(* Logix 5000 project; controller PLC vendor 1 type 14 code 155 rev 30.14; software revision 30.01 *)

TASK MainTask (continuous, watchdog 500 ms) : MainProgram

MODULES
   Local : vendor 1 type 14 code 155 (PointIO 0, rev 30.14)
      Encoder_Conveyor : vendor 1 type 37 code 52 (Ethernet 192.168.100.195, rev 1.1, MotionDiagnostics RPI 1 ms, MotionSync RPI 4 ms)
      Servo_Bridge_Shift : vendor 1 type 37 code 49 (Ethernet 192.168.100.194, rev 7.1, MotionSync RPI 4 ms, MotionDiagnostics RPI 1 ms)
      Rack_0_Slot_2 : 1734-IB8 (PointIO 2, rev 3.1, Input RPI 20 ms)
           Local:2:I.Data.0   // Slot 2 Input 0
           Local:2:I.Data.1   // Slot 2 Input 1
           Local:2:I.Data.2   // Slot 2 Input 2
           Local:2:I.Data.3   // Slot 2 Input 3
           Local:2:I.Data.4   // Slot 2 Input 4
           Local:2:I.Data.5   // Slot 2 Input 5
           Local:2:I.Data.6   // Slot 2 Input 6
           Local:2:I.Data.7   // Slot 2 Input 7
      Rack_0_Slot_3 : 1734-OB8 (PointIO 3, rev 3.1, Output RPI 20 ms)
           Local:3:O.Data.0   // Slot 3 Output 0
           Local:3:O.Data.1   // Slot 3 Output 1
           Local:3:O.Data.2   // Slot 3 Output 2
           Local:3:O.Data.3   // Slot 3 Output 3
           Local:3:O.Data.4   // Slot 3 Output 4
           Local:3:O.Data.5   // Slot 3 Output 5
           Local:3:O.Data.6   // Slot 3 Output 6
           Local:3:O   // Slot 3 Output
      Discrete_IO : Embedded (PointIO 1, rev 30.11, Output RPI 20 ms)
           Local:1:O   // Slot 1 Output
           Local:1:I.Data.0   // Slot 0 Input 0
           Local:1:I.Data.1   // Slot 0 Input 1
           Local:1:I.Data.10   // Slot 0 Input 10
           Local:1:I.Data.11   // Slot 0 Input 11
           Local:1:I.Data.12   // Slot 0 Input 12
           Local:1:I.Data.13   // Slot 0 Input 13
           Local:1:I.Data.14   // Slot 0 Input 14
           Local:1:I.Data.15   // Slot 0 Input 15
           Local:1:I.Data.2   // Slot 0 Input 2
           Local:1:I.Data.3   // Slot 0 Input 3
           Local:1:I.Data.4   // Slot 0 Input 4
           Local:1:I.Data.5   // Slot 0 Input 5
           Local:1:I.Data.6   // Slot 0 Input 6
           Local:1:I.Data.7   // Slot 0 Input 7
           Local:1:I.Data.8   // Slot 0 Input 8
           Local:1:I.Data.9   // Slot 0 Input 9
      Rack_0_Slot_4 : 1734-OB8 (PointIO 4, rev 3.1, Output RPI 20 ms)
           Local:4:O   // Slot 4 Output
END_MODULES

TYPE Axis_MC_R3b :
STRUCT
   Auto_Enable : BOOL;
   Direction_Fwd : BOOL;
   Direction_Rev : BOOL;
   Direction_Fwd_DINT : DINT;
   Direction_Rev_DINT : DINT;
   Multiplier_Distance : REAL;
   Multiplier_Speed : REAL;
   Multiplier_Acc_Dec : REAL;
   Distance_Home_Offset : REAL;
   Distance_Row_to_Row : REAL;
   Distance_First_Row : REAL;
   Distance_Flight_to_Flight : REAL;
   Number_of_Rows : REAL;
   Speed_Homing : REAL;
   Speed_Jog_FWD : REAL;
   Speed_Jog_REV : REAL;
   Speed_Prime : REAL;
   Speed_Cleaning : REAL;
   Speed_Auto_FWD : REAL;
   Speed_Auto_REV : REAL;
   Accel_Homing : REAL;
   Accel_Jog : REAL;
   Accel_Prime : REAL;
   Accel_Auto : REAL;
   Accel_Raw : REAL;
   Accel_Scaled : REAL;
   Decel_Estop : REAL;
   Decel_Homing : REAL;
   Decel_Jog : REAL;
   Decel_Prime : REAL;
   Decel_Auto : REAL;
   Decel_Raw : REAL;
   Decel_Scaled : REAL;
   Status_Faulted : BOOL;
   Status_Fault_Code : DINT;
   Status_Homed : BOOL;
   Status_Homing : BOOL;
   Status_Raw_Position : DINT;
   Status_Scaled_Position : REAL;
   Status_Jogging : BOOL;
   Status_Jogging_Stopped_OS : BOOL;
   Status_In_Motion : BOOL;
   Status_In_Motion_OS : BOOL;
   Status_Stopped : BOOL;
   Status_Stopped_OS : BOOL;
   Status_Safe_to_Move : BOOL;
   HMI_PB_Jog_FWD : BOOL;
   HMI_PB_Jog_REV : BOOL;
   Jog_FWD : BOOL;
   Jog_REV : BOOL;
   Jog_FWD_OS : BOOL;
   Jog_REV_OS : BOOL;
   HMI_PB_Home_Servo : BOOL;
   HMI_PB_Home_Servo_OS : BOOL;
   Homing_Needed_Next_Move : BOOL;   // Registration needed during next long move
   Homing_Needed_Now : BOOL;   // Registration needed after e-stop
   Homing_Counter : COUNTER;   // Registration counter for cycles before homing or registration needed
   Homing_Counter_DN_OS : BOOL;
   Homing_Timer_Step : TIMER[10];
   Homing_Sensor_Active_OS : BOOL;
   Homing_Sensor_Deactive_OS : BOOL;
   Homing_Failure : BOOL;
   Timer_Jog_FWD_Delay : TIMER;
   Timer_Jog_REV_Delay : TIMER;
   Timer_Servo_Safe_to_Move : TIMER;
   Overtravel_Fwd_Active_OS : BOOL;
   Overtravel_Fwd_Deactive_OS : BOOL;
   Overtravel_Rev_Active_OS : BOOL;
   Overtravel_Rev_Deactive_OS : BOOL;
   Overtravel_Front_Active_OS : BOOL;
   Overtravel_Front_Deactive_OS : BOOL;
   Overtravel_Rear_Active_OS : BOOL;
   Overtravel_Rear_Deactive_OS : BOOL;
   Cam_M_Offset : DINT;
   Cam_S_Offset : DINT;
   Cam_M_Scaling : DINT;
   Cam_S_Scaling : DINT;
   OS : DINT[2];
   MSO : MOTION_INSTRUCTION;
   MSF : MOTION_INSTRUCTION;
   MASR : MOTION_INSTRUCTION;
   MAFR : MOTION_INSTRUCTION;
   MAJ : MOTION_INSTRUCTION[10];
   MAJ_DIRECTION : DINT[10];
   MAJ_SPEED : REAL[10];
   MAJ_ACC : REAL[10];
   MAJ_DEC : REAL[10];
   MAM : MOTION_INSTRUCTION[10];
   MAM_TYPE : DINT[10];
   MAM_DISTANCE : REAL[10];
   MAM_SPEED : REAL[10];
   MAM_ACC : REAL[10];
   MAM_DEC : REAL[10];
   MAS : MOTION_INSTRUCTION[10];
   MAS_DEC : REAL[10];
   MAH : MOTION_INSTRUCTION[5];
   MCD : MOTION_INSTRUCTION[10];
   MRP : MOTION_INSTRUCTION;
   MGS : MOTION_INSTRUCTION;
   MGSD : MOTION_INSTRUCTION;
   MGSR : MOTION_INSTRUCTION;
   MGSP : MOTION_INSTRUCTION;
   MAG : MOTION_INSTRUCTION[5];
   MAG_DIRECTION : DINT[5];
   MAG_TYPE : DINT[5];
   MAG_DISTANCE : REAL[5];
   MAG_SPEED : REAL[5];
   MAG_ACC : REAL[5];
   MAG_DEC : REAL[5];
   MAG_RATIO : REAL[5];
   MAG_S_COUNTS : DINT[5];
   MAG_M_COUNTS : DINT[5];
END_STRUCT
END_TYPE

TYPE Denester_R2b :
STRUCT
   HMI_Auger_VFD_Jog : BOOL;
   HMI_Trigger : BOOL;
   HMI_Trigger_OS : BOOL;
   Trigger : BOOL;
   Trigger_OS : BOOL;
   Auger_Direction_Fwd : BOOL;
   Auger_Direction_Rev : BOOL;
   Auger_VFD_Run : BOOL;
   Auger_VFD_Jog : BOOL;
   Auger_VFD_Speed_Auto : REAL;
   Auger_VFD_Speed_Jog : REAL;
   Auger_Prox_OS : BOOL;
   Status_Ready : BOOL;
   Status_Done : BOOL;
   Status_Done_OS : BOOL;
   Timer_Auger_Run_Delay : TIMER;
   Low_Cups_OS : BOOL;
   Low_Cups_Warning : BOOL;
   Timer_Trigger_Delay : TIMER;
   Timer_Trigger_Duration : TIMER;
   OS : DINT;
END_STRUCT
END_TYPE

TYPE Depositor_R2b :
STRUCT
   HMI_Trigger_Deposit : BOOL;
   HMI_Trigger_Deposit_OS : BOOL;
   Prime_Trigger_Deposit_OS : BOOL;
   Trigger_Deposit : BOOL;
   Trigger_Deposit_OS : BOOL;
   Piston_Deposit : DINT;   // Product Piston deposit
   Piston_Suction : DINT;   // Product Piston suction
   Product_Valve_Deposit : DINT;   // Product Valve deposit position
   Spout_Open : DINT;   // Open Spout
   Dive_Down : DINT;
   Dive_Up : DINT;
   Status_Suction_Complete : BOOL;
   Status_Suction_Complete_OS : BOOL;
   Status_Deposit_Complete : BOOL;
   Status_Deposit_Complete_OS : BOOL;
   Status_Done : BOOL;
   Status_Done_OS : BOOL;
   Status_Ready : BOOL;
   Timer_Blowoff_Delay : TIMER;
   Timer_Blowoff_Duration : TIMER;
   Timer_Dive_Delay : TIMER;
   Timer_Dive_Duration : TIMER;
   Timer_Dive_Timeout : TIMER;
   Timer_Trigger_Duration : TIMER;
   Timer_Trigger_Delay : TIMER;
   Timer_Prime : TIMER;
   Timer_Shift_Delay_Suction : TIMER;
   Timer_Shift_Delay_Deposit : TIMER;
   Timer_Spout_Timeout : TIMER;
   OS : DINT;
END_STRUCT
END_TYPE

TYPE Forces_R2b :
STRUCT
   DI_0 : DINT;   // INPUT FORCE
   DI_1 : DINT;   // INPUT FORCE
   DI_2 : DINT;   // INPUT FORCE
   DI_3 : DINT;   // INPUT FORCE
   DI_4 : DINT;   // INPUT FORCE
   DI_5 : DINT;   // INPUT FORCE
   DO_0 : DINT;   // OUTPUT FORCE
   DO_1 : DINT;   // OUTPUT FORCE
   DO_2 : DINT;   // OUTPUT FORCE
   DO_3 : DINT;   // OUTPUT FORCE
   DO_4 : DINT;   // OUTPUT FORCE
   DO_5 : DINT;   // OUTPUT FORCE
   DO_6 : DINT;   // OUTPUT FORCE
   DO_7 : DINT;   // OUTPUT FORCE
   DO_8 : DINT;   // OUTPUT FORCE
   DO_9 : DINT;   // OUTPUT FORCE
   DO_10 : DINT;   // OUTPUT FORCE
   R_DO_0 : DINT;   // OUTPUT FORCE
   R_DO_1 : DINT;   // OUTPUT FORCE
   R_DO_2 : DINT;   // OUTPUT FORCE
   R_DO_3 : DINT;   // OUTPUT FORCE
   R_DO_4 : DINT;   // OUTPUT FORCE
   R_DO_5 : DINT;   // OUTPUT FORCE
END_STRUCT
END_TYPE

TYPE IO_R2a :
STRUCT
   DI_0 : DINT;
   DI_1 : DINT;
   DI_2 : DINT;
   DI_3 : DINT;
   DI_4 : DINT;
   DI_5 : DINT;
   DI_6 : DINT;
   DI_7 : DINT;
   DI_8 : DINT;
   DI_9 : DINT;
   DI_10 : DINT;
   DO_0 : DINT;
   DO_1 : DINT;
   DO_2 : DINT;
   DO_3 : DINT;
   DO_4 : DINT;
   DO_5 : DINT;
   DO_6 : DINT;
   DO_7 : DINT;
   DO_8 : DINT;
   DO_9 : DINT;
   DO_10 : DINT;
   R_DI_0 : DINT;
   R_DI_1 : DINT;
   R_DI_2 : DINT;
   R_DI_3 : DINT;
   R_DI_4 : DINT;
   R_DI_5 : DINT;
   R_DO_0 : DINT;
   R_DO_1 : DINT;
   R_DO_2 : DINT;
   R_DO_3 : DINT;
   R_DO_4 : DINT;
   R_DO_5 : DINT;
END_STRUCT
END_TYPE

TYPE Login_R2a :
STRUCT
   User : DINT;
   User_Logged_In : DINT;
   User_New : DINT;
   User_Active : BOOL;
   No_Access : BOOL;
   Password_Entered : DINT;
   Password_New : DINT;
   Password_Old : DINT;
   Password_Admin : DINT;
   Password_Maint : DINT;
   Password_Lead : DINT;
   Password_HBTech : DINT;
   Password_Temp : DINT;
   Password_Backdoor : DINT;
   Password_Oper : DINT;
   PB_Reset_Passwords : BOOL;
   PB_Change_Password : BOOL;
   PB_Change_Password_Yes : BOOL;
   PB_Change_Password_No : BOOL;
   PB_Logout : BOOL;
   Auto_Logout_Minutes : INT;
   Timer_Auto_Logout : TIMER;
   Timer_Reset_Delay : TIMER;
   Timer_Password_Change_Confirm : TIMER;
   Timer_Password_Change_Timeout : TIMER;
   Visible_New_Password : BOOL;
   Visible_Change_Password : BOOL;
   Visible_Change_Confirm : BOOL;
   Visible_Password_Changed : BOOL;
END_STRUCT
END_TYPE

TYPE NCNF_Arrays_R2a :
STRUCT
   Bitshift : DINT[4];
END_STRUCT
END_TYPE

TYPE NCNF_R2a :
STRUCT
   Flight_Detect_OS_Rising : BOOL;   // FLIGHT DETECT RISING OS
   Flight_Detect_OS_Falling : BOOL;   // FLIGHT DETECT FALLING OS
   Target_Detected : BOOL[32];   // NC/NF TARGET DETECTED
   Lane : NCNF_Arrays_R2a[10];   // NC/NF BITSHIFTS
   Bitshift_Control : CONTROL[10];   // NC/NF BITSHIFT CONTROLS
   HMI_PB_Reset : BOOL;   // NC/NF HMI BITSHIFT RESET
   HMI_PB_Fill : BOOL;   // NC/NF HMI BITSHIFT FILL
   HMI_PB_Bypass : BOOL;   // NC/NF HMI BITSHIFT BYPASS
   Timer_Flight_Detect_OFF : TIMER;
END_STRUCT
END_TYPE

TYPE Rates_R2b :
STRUCT
   HMI_PB_Reset_Counter : BOOL;
   Counter_Cycle : COUNTER;
   Counter_Total : COUNTER;
   Timer_CPM_Minute : TIMER;
   Timer_CPM_Seconds : DINT;
   Timer_Cycle_Time : TIMER;
   Cycle_Time : DINT;
   CPM_Current : DINT;
   CPM_Previous : DINT;
   PPM_Current : DINT;
   PPM_Previous : DINT;
   Rows_Per_Pan : DINT;
   Total_Count : DINT;
END_STRUCT
END_TYPE

TYPE Recipe_R2c :
STRUCT
   Active_Recipe_Num : DINT;
   Active_Recipe_Name : STRING;
   Active_Recipe : DINT[15];
   Selected_Recipe_Num : DINT;
   Selected_Recipe_Name : STRING;
   Selected_Recipe : DINT[15];
   Selected_Recipe_Edit_Num : DINT;
   Previous_Selected_Recipe_Num : DINT;
   Indirect_Recipe_Selected : DINT;
   Indirect_Recipe_Selected_Edit : DINT;
   Recipe_Changed_OS : BOOL;
   Load_Selected_Recipe_Num : DINT;
   Saveas_Source_Recipe_Num : DINT;
   Saveas_Target_Recipe_Num : DINT;
   HMI_PB_Load : BOOL;
   HMI_PB_Save : BOOL;
   HMI_PB_Saveas : BOOL;
   HMI_PB_Rename : BOOL;
   Timer_Load : TIMER;
   Timer_Save : TIMER;
   Timer_Saveas : TIMER;
   Names_Pointer : DINT;
   Names_Pointer_Temp : DINT;
   Names_New_Name : STRING;
   Names_Old_Name : STRING;
END_STRUCT
END_TYPE

TYPE Sequencer_R2a :
STRUCT
   Step : DINT;   // Current Step
   Step_OS : BOOL[256];   // Current Step OS
   Timer : TIMER[256];   // Current Step Timer
   OS : BOOL[256];   // OS
END_STRUCT
END_TYPE

TYPE System_R2e :   // System
STRUCT
   HMI_Current_Screen : DINT;
   HMI_Forced_Screen : DINT;
   HMI_PB_Estop_Reset : BOOL;
   HMI_PB_Start : BOOL;
   HMI_PB_Stop : BOOL;
   HMI_PB_Prime : BOOL;
   HMI_PB_Prime_OS : BOOL;
   HMI_PB_Auto : BOOL;
   HMI_PB_Auto_OS : BOOL;
   HMI_PB_Clean : BOOL;
   HMI_PB_Clean_OS : BOOL;
   HMI_PB_Clear_Alarms : BOOL;
   HMI_PB_Silence_Alarms : BOOL;
   HMI_PB_Home_Servos : BOOL;
   HMI_PB_Home_Servos_OS : BOOL;
   HMI_PB_Off : BOOL;
   HMI_PB_Off_OS : BOOL;
   HMI_PB_Wipe_Screen_Reset : BOOL;
   HMI_PB_Recipe_Initialize : BOOL;
   HMI_Visible_PB : BOOL;
   HMI_Visible_Estop_Reset : BOOL;
   HMI_Visible_Home_Servos : BOOL;
   HMI_Visible_Clear_Alarms : BOOL;
   HMI_Visible_Silence_Alarms : BOOL;
   Local_PB_Start : BOOL;
   Local_PB_Stop : BOOL;
   Local_Estop_Reset : BOOL;
   Estop_Reset_Enabled : BOOL;
   Timer_Starting : TIMER;
   Timer_Starting_TT_OS : BOOL;
   Timer_Starting_DN_OS : BOOL;
   Timer_Stopping : TIMER;
   Timer_Stopping_EN_OS : BOOL;
   Timer_Stopping_DN_OS : BOOL;
   Timer_Estop_Not_OK : TIMER;
   Timer_Estop_Not_OK_TT_OS : BOOL;
   Timer_Estop_Not_OK_DN_OS : BOOL;
   Timer_EStop_Reset : TIMER;
   Timer_Estop_OK : TIMER;
   Timer_Estop_OK_TT_OS : BOOL;
   Timer_Estop_OK_DN_OS : BOOL;
   Timer_Power_Up : TIMER;
   Timer_Power_Up_OS : BOOL;
   Timer_Alarm_Timeout : TIMER;
   Timer_Alarm_Timeout_OS : BOOL;
   Timer_Flasher_Slow_On : TIMER;
   Timer_Flasher_Slow_Off : TIMER;
   Timer_Flasher_Fast_On : TIMER;
   Timer_Flasher_Fast_Off : TIMER;
   Timer_Servos_Home : TIMER;
   Timer_Alarm_Horn : TIMER;
   Timer_Wipe_Screen : TIMER;
   Timer_Screen_Force : TIMER;
   Mode_Auto : BOOL;
   Mode_Off : BOOL;
   Mode_Prime : BOOL;
   Mode_Clean : BOOL;
   Mode_Integer : DINT;
   Mode_Changed_OS : BOOL;
   Status_EStop_Active : BOOL;
   Status_Estop_OK : BOOL;
   Status_Estop_OK_OS : BOOL;
   Status_Estop_NOT_OK : BOOL;
   Status_Estop_NOT_OK_OS : BOOL;
   Status_Alarm : BOOL;
   Status_Alarm_OS : BOOL;
   Status_New_Alarm : BOOL;
   Status_Warning : BOOL;
   Status_DINT : DINT;   // \
   Servos_Home : BOOL;
   Servos_Home_OS : BOOL;
   Servos_Homed : BOOL;
   Servos_Homed_OS : BOOL;
   Servos_Homing_Requested : BOOL;
   Servos_Homing : BOOL;
   Servos_Homing_OS : BOOL;
   Servos_OK : BOOL;
   Always_ON_Bit : BOOL;
   Always_OFF_Bit : BOOL;
   Test_Bits : DINT;
   Comms_Scan_Timer : TIMER;
   Comms_Scan_Counter : DINT;
END_STRUCT
END_TYPE

VAR_GLOBAL   (* controller tags *)
   Alarm_Timer : TIMER[2,32] := ([0,1].PRE := 1000, [0,2].PRE := 5, [0,3].PRE := 5, [0,4].PRE := 5, [0,5].PRE := 10, [0,6].PRE := 100, [0,7].PRE := 500, [0,8].PRE := 5000, [0,9].PRE := 7500, [0,10].PRE := 500, [0,11].PRE := 20000, [0,12].PRE := 5, [0,13].PRE := 5, [0,14].PRE := 5, [0,15].PRE := 5, [0,16].PRE := 5, [0,17].PRE := 1000, [0,18].PRE := 2000, [0,19].PRE := 100, [0,20].PRE := 20000, [0,21].PRE := 20000, [0,22].PRE := 100, [0,23].PRE := 100);
   Alarm_Word_Compare : DINT[3];
   Alarm_Word_Current : DINT[3];
   Alarm_Word_New : DINT[3];
   Alarm_Word_Previous : DINT[3];
   always_open : BOOL;
   Bridge_Timer_Gearing_Delay : TIMER := (PRE := 30);
   Bridge_Timer_Gearing_Delay_DN_OS : BOOL;
   Bridge_Timer_Gearing_Duration : TIMER;
   Bridge_Timer_Gearing_Duration_DN_OS : BOOL;
   Bypass_Encoder : BOOL;
   Denester : Denester_R2b := (Timer_Trigger_Delay.PRE := 5, Timer_Trigger_Duration.PRE := 40);
   Denester_Flight_Counter : COUNTER := (PRE := 1);
   Denester_index_counter : COUNTER := (PRE := 4, ACC := 2);
   Depositor : Depositor_R2b := (Timer_Blowoff_Delay.PRE := 20, Timer_Blowoff_Duration.PRE := 200, Timer_Dive_Delay.PRE := 5, Timer_Dive_Duration.PRE := 1095, Timer_Trigger_Delay.PRE := 25, Timer_Prime.PRE := 1000, Timer_Spout_Timeout.PRE := 1500);
   Depositor_Bridge_Up : BOOL;
   Encoder_Conveyor : AXIS_CIP_DRIVE;
   equal_to_20 : BOOL;
   FORCE_GO_SIGNAL : BOOL;
   FORCE_TRIGGER : BOOL;
   Forces : Forces_R2b := (DO_3 := 8);
   HMI_Enable_Denester : BOOL := 1;
   homing_timeout : TIMER := (PRE := 20000);
   IO : IO_R2a := (DI_1 := 33228, DI_2 := 32, DO_1 := 34, DO_3 := 8);
        .DI_2.0   // SPARE
        .DI_2.1   // BRIDGE UP PROX
        .DI_2.2   // BRIDGE OVERTRAVEL PROX
        .DI_2.3   // BRIDGE HOME PROX
        .DI_2.4   // SPARE
        .DI_2.5   // SPARE
        .DI_2.6   // SPARE
        .DI_2.7   // SPARE
        .DO_1.0   // STACK LIGHT HORN
        .DO_1.1   // STACK LIGHT GREEN
        .DO_1.10   // FILLER SPOUT #3 TRIGGER
        .DO_1.11   // FILLER SPOUT #4 TRIGGER
        .DO_1.12   // FILLER SPOUT #5 TRIGGER
        .DO_1.13   // FILLER SPOUT #6 TRIGGER
        .DO_1.14   // FILLER SPOUT #7 TRIGGER
        .DO_1.15   // FILLER SPOUT #8 TRIGGER
        .DO_1.2   // STACK LIGHT AMBER
        .DO_1.3   // STACK LIGHT RED
        .DO_1.4   // DONE SIGNAL TO CUSTOMER
        .DO_1.5   // PLC E-STOP RESET
        .DO_1.6   // READY SIGNAL TO CUSTOMER
        .DO_1.7   // DENESTER TRIGGER
        .DO_1.8   // FILLER SPOUT #1 TRIGGER
        .DO_1.9   // FILLER SPOUT #2 TRIGGER
        .DO_3.0   // BRIDGE DOWN SPOUTS #1-4
        .DO_3.1   // BRIDGE UP SPOUTS #1-4
        .DO_3.2   // BLOWOFF SPOUTS #1-4
        .DO_3.3   // SPOUT #1 OPEN
        .DO_3.4   // SPOUT #2 OPEN
        .DO_3.5   // SPOUT #3 OPEN
        .DO_3.6   // SPOUT #4 OPEN
        .DO_3.7   // SPARE
        .DO_4.0   // BRIDGE DOWN SPOUTS #5-8
        .DO_4.1   // BRIDGE UP SPOUTS #5-8
        .DO_4.2   // BLOWOFF SPOUTS #5-8
        .DO_4.3   // SPOUT #5 OPEN
        .DO_4.4   // SPOUT #6 OPEN
        .DO_4.5   // SPOUT #7 OPEN
        .DO_4.6   // SPOUT #8 OPEN
        .DO_4.7   // SPARE
        .DI_1.0   // SPARE
        .DI_1.1   // SPARE
        .DI_1.10   // FILLER PRIME MODE ACTIVE
        .DI_1.11   // E-STOP PRESSED 1-HOLE UPSTREAM
        .DI_1.12   // ULMA GO SIGNAL/ FLIGHT DETECT
        .DI_1.13   // ULMA RUNNING RELAY
        .DI_1.14   // NC/NF SENSOR LANE #0
        .DI_1.15   // NC/NF SENSOR LANE #1
        .DI_1.2   // AIR PRESSURE SWITCH
        .DI_1.3   // E-STOP OK
        .DI_1.4   // E-STOP PRESSED MAIN
        .DI_1.5   // E-STOP PRESSED 1-HOLE DOWNSTREAM
        .DI_1.6   // UPSTREAM DOOR
        .DI_1.7   // DOWNSTREAM DOOR
        .DI_1.8   // DOCKING SAFETY SENSOR
        .DI_1.9   // FILLER DONE/READY
   Login : Login_R2a := (Password_Admin := 111, Password_Maint := 222, Password_Lead := 333, Password_HBTech := 32767, Password_Temp := 555, Password_Backdoor := 80808, Password_Oper := 444, Auto_Logout_Minutes := 60, Timer_Auto_Logout.PRE := 3600000);
        .User   // Login User 1 = ADMIN 2 = MAINT 3 = LEAD 4 = OPER 5 = TEMP 6 = BACKDOOR 7 = HBTECH
        .User_Logged_In   // Login User Logged In
        .Password_Entered   // Login Password Entered
   MV_conveyor_moving : BOOL;
   MV_conveyor_stopped : BOOL;
   MV_Encoder_Stop_Threshold : DINT;
   MV_Encoder_Stop_Value : REAL := 0.3;
   MV_Encoder_Stop_Value2 : REAL := 0.2;
   mv_index_counter : COUNTER := (PRE := 15, ACC := 5);
   MV_indexes : DINT := 4;
   MV_Rate : DINT := 100;
   MV_total_indexes : COUNTER := (PRE := 100, ACC := 343, DN := 1);
   NC_NF : NCNF_R2a := (Target_Detected[1] := 1, Lane[0].Bitshift[0] := 2147483647, Lane[0].Bitshift[1] := 2147483647, Lane[0].Bitshift[2] := 2147483647, Lane[0].Bitshift[3] := 2147483647, Lane[1].Bitshift[0] := 2147483647, Lane[1].Bitshift[1] := 2147483647, Lane[1].Bitshift[2] := 2147483647, Lane[1].Bitshift[3] := 2147483647, Bitshift_Control[0].LEN := 4, Bitshift_Control[0].UL := 1, Bitshift_Control[1].LEN := 4, Bitshift_Control[1].UL := 1, HMI_PB_Bypass := 1);   // NC/NF BITSHIFTS
        .Flight_Detect_OS_Rising   // Flight Detect One Shot Rising
        .Flight_Detect_OS_Falling   // Flight Detect One Shot Falling
   OS : INT[10] := ([0] := 268, [1] := 42, [2] := 28356, [3] := 2114, [4] := 6176, [5] := 19966, [6] := -32768);
        [0].15   // DUMMY TEST BIT
        [2].2   // SUTEY
        [2].5   // TEST BIT
        [3].13   // IGNORE
        [2].3   // SUTEY
        [5].0   // OS to position Bridge for CIP
        [7].0   // TEST BIT
        [3].2   // SUTEY
   Rates : Rates_R2b := (Counter_Cycle.PRE := 1000, Counter_Total.PRE := 10000000, Counter_Total.ACC := 701468, Timer_CPM_Minute.PRE := 60000, Timer_CPM_Minute.ACC := 3755, Timer_CPM_Minute.EN := 1, Timer_CPM_Minute.TT := 1, Timer_CPM_Seconds := 3, Timer_Cycle_Time.ACC := 1, Timer_Cycle_Time.EN := 1, Timer_Cycle_Time.DN := 1, Cycle_Time := 1);
   Recipe : Recipe_R2c := (Selected_Recipe_Num := 1, Selected_Recipe_Edit_Num := 22, Previous_Selected_Recipe_Num := 1);
        .Active_Recipe[0].0   // Active Recipe VFD Conveyor ON/OFF
   Recipe_Names : STRING[23] := ([1] := ' 2ZOG AU', [2] := 'ERICEP2 ', [3] := 'ERICEP3 ', [4] := 'ERICEP4 ', [5] := 'ERICEP5 ', [6] := 'ERICEP6 ', [7] := 'ERICEP7 ', [8] := 'ERICEP8 ', [9] := 'ERICEP9 ', [10] := 'ERICEP1  0', [11] := 'ERICEP1  1', [12] := 'ERICEP1  2', [13] := 'ERICEP1  3', [14] := 'ERICEP1  4', [15] := 'ERICEP1  5', [16] := 'ERICEP1  6', [17] := 'ERICEP1  7', [18] := 'ERICEP1  8', [19] := 'ERICEP1  9', [20] := 'ERICEP2  0', [21] := 'ETTS', [22] := 'ETTS');
   Recipe_Setpoints_DINT : DINT[23,20] := ([0,0] := 55, [0,1] := 56, [0,2] := 56, [0,3] := 15, [0,7] := 51, [0,8] := 60, [0,12] := 52, [0,13] := 60, [1,0] := 63, [1,1] := 56, [1,2] := 56, [1,3] := 15, [1,7] := 51, [1,8] := 60, [1,12] := 52, [1,13] := 60, [2,0] := 63, [2,1] := 56, [2,2] := 56, [2,3] := 15, [2,7] := 51, [2,8] := 60, [2,12] := 52, [2,13] := 60, [3,0] := 63, [3,1] := 56, [3,2] := 56, [3,3] := 15, [3,7] := 51, [3,8] := 60, [3,12] := 52, [3,13] := 60, [4,0] := 63, [4,1] := 56, [4,2] := 56, [4,3] := 15, [4,7] := 51, [4,8] := 60, [4,12] := 52, [4,13] := 60, [5,0] := 63, [5,1] := 56, [5,2] := 56, [5,3] := 15, [5,7] := 51, [5,8] := 60, [5,12] := 52, [5,13] := 60, [6,0] := 63, [6,1] := 56, [6,2] := 56, [6,3] := 15, [6,7] := 51, [6,8] := 60, [6,12] := 52, [6,13] := 60, [7,0] := 63, [7,1] := 56, [7,2] := 56, [7,3] := 15,
        [7,7] := 51, [7,8] := 60, [7,12] := 52, [7,13] := 60, [8,0] := 63, [8,1] := 56, [8,2] := 56, [8,3] := 15, [8,7] := 51, [8,8] := 60, [8,12] := 52, [8,13] := 60, [9,0] := 63, [9,1] := 56, [9,2] := 56, [9,3] := 15, [9,7] := 51, [9,8] := 60, [9,12] := 52, [9,13] := 60, [10,0] := 63, [10,1] := 56, [10,2] := 56, [10,3] := 15, [10,7] := 51, [10,8] := 60, [10,12] := 52, [10,13] := 60, [11,0] := 63, [11,1] := 56, [11,2] := 56, [11,3] := 15, [11,7] := 51, [11,8] := 60, [11,12] := 52, [11,13] := 60, [12,0] := 63, [12,1] := 56, [12,2] := 56, [12,3] := 15, [12,7] := 51, [12,8] := 60, [12,12] := 52, [12,13] := 60, [13,0] := 63, [13,1] := 56, [13,2] := 56, [13,3] := 15, [13,7] := 51, [13,8] := 60, [13,12] := 52, [13,13] := 60, [14,0] := 63, [14,1] := 56, [14,2] := 56, [14,3] := 15, [14,7] := 51, [14,8] := 60, [14,12] := 52, [14,13] := 60,
        [15,0] := 63, [15,1] := 56, [15,2] := 56, [15,3] := 15, [15,7] := 51, [15,8] := 60, [15,12] := 52, [15,13] := 60, [16,0] := 63, [16,1] := 56, [16,2] := 56, [16,3] := 15, [16,7] := 51, [16,8] := 60, [16,12] := 52, [16,13] := 60, [17,0] := 63, [17,1] := 56, [17,2] := 56, [17,3] := 15, [17,7] := 51, [17,8] := 60, [17,12] := 52, [17,13] := 60, [18,0] := 63, [18,1] := 56, [18,2] := 56, [18,3] := 15, [18,7] := 51, [18,8] := 60, [18,12] := 52, [18,13] := 60, [19,0] := 63, [19,1] := 56, [19,2] := 56, [19,3] := 15, [19,7] := 51, [19,8] := 60, [19,12] := 52, [19,13] := 60, [20,0] := 63, [20,1] := 56, [20,2] := 56, [20,3] := 15, [20,7] := 51, [20,8] := 60, [20,12] := 52, [20,13] := 60, [21,0] := 63, [21,1] := 56, [21,2] := 56, [21,3] := 15, [21,7] := 51, [21,8] := 60, [21,12] := 52, [21,13] := 60, [22,0] := 63, [22,1] := 56, [22,2] := 56, [22,3] := 15,
        [22,7] := 51, [22,8] := 60, [22,12] := 52, [22,13] := 60);
        [0,0]   // Recipe Bools
        [0,0].0   // Recipe Depositor On/Off
        [0,0].1   // Recipe Bridge Dive On/Off
        [0,0].2   // Recipe Bridge Shift On/Off
        [0,0].3   // Recipe Blowoff On/Off
        [0,0].4   // Recipe Orbit B On/Off
        [0,0].5   // Recipe Filler A On/Off
        [0,0].6   // Filler A Level Control On/Off
        [0,0].7   // Filler B Level Control On/Off
        [0,12]   // Filler B Suction Velocity
        [0,13]   // Filler B Deposit Velocity
        [0,1]   // Flighted Conveyor Speed
        [0,2]   // Overrrunning Conveyor Speed
        [0,7]   // Filler A Suction Velocity
        [0,8]   // Filler A Deposit Velocity
   Recipe_Setpoints_DINT_Temp : DINT[20] := ([0] := 63, [1] := 56, [2] := 56, [3] := 15, [7] := 51, [8] := 60, [12] := 52, [13] := 60);
   Recipe_Setpoints_REAL : REAL[23,20] := ([0,0] := 5.0, [0,1] := 0.7, [0,2] := 20.0, [0,3] := 200.0, [0,4] := 5.0, [0,5] := 1095.0, [0,6] := 51.0, [0,8] := 100.0, [0,9] := 200.0, [0,10] := 5.0, [0,14] := 7.5, [0,15] := 10.0, [1,0] := 5.0, [1,1] := 0.7, [1,2] := 400.0, [1,3] := 75.0, [1,4] := 5.0, [1,5] := 800.0, [1,6] := 51.0, [1,8] := 100.0, [1,9] := 200.0, [1,14] := 7.5, [1,15] := 10.0, [2,0] := 5.0, [2,1] := 0.7, [2,2] := 400.0, [2,3] := 75.0, [2,4] := 5.0, [2,5] := 800.0, [2,6] := 51.0, [2,8] := 100.0, [2,9] := 200.0, [2,14] := 7.5, [2,15] := 10.0, [3,0] := 5.0, [3,1] := 0.7, [3,2] := 400.0, [3,3] := 75.0, [3,4] := 5.0, [3,5] := 800.0, [3,6] := 51.0, [3,8] := 100.0, [3,9] := 200.0, [3,14] := 7.5, [3,15] := 10.0, [4,0] := 5.0, [4,1] := 0.7, [4,2] := 400.0, [4,3] := 75.0, [4,4] := 5.0, [4,5] := 800.0, [4,6] := 51.0, [4,8] := 100.0, [4,9] := 200.0, [4,14] := 7.5, [4,15] := 10.0, [5,0] := 5.0, [5,1] := 0.7, [5,2] := 400.0, [5,3] := 75.0,
        [5,4] := 5.0, [5,5] := 800.0, [5,6] := 51.0, [5,8] := 100.0, [5,9] := 200.0, [5,14] := 7.5, [5,15] := 10.0, [6,0] := 5.0, [6,1] := 0.7, [6,2] := 400.0, [6,3] := 75.0, [6,4] := 5.0, [6,5] := 800.0, [6,6] := 51.0, [6,8] := 100.0, [6,9] := 200.0, [6,14] := 7.5, [6,15] := 10.0, [7,0] := 5.0, [7,1] := 0.7, [7,2] := 400.0, [7,3] := 75.0, [7,4] := 5.0, [7,5] := 800.0, [7,6] := 51.0, [7,8] := 100.0, [7,9] := 200.0, [7,14] := 7.5, [7,15] := 10.0, [8,0] := 5.0, [8,1] := 0.7, [8,2] := 400.0, [8,3] := 75.0, [8,4] := 5.0, [8,5] := 800.0, [8,6] := 51.0, [8,8] := 100.0, [8,9] := 200.0, [8,14] := 7.5, [8,15] := 10.0, [9,0] := 5.0, [9,1] := 0.7, [9,2] := 400.0, [9,3] := 75.0, [9,4] := 5.0, [9,5] := 800.0, [9,6] := 51.0, [9,8] := 100.0, [9,9] := 200.0, [9,14] := 7.5, [9,15] := 10.0, [10,0] := 5.0, [10,1] := 0.7, [10,2] := 400.0, [10,3] := 75.0, [10,4] := 5.0, [10,5] := 800.0, [10,6] := 51.0, [10,8] := 100.0, [10,9] := 200.0,
        [10,14] := 7.5, [10,15] := 10.0, [11,0] := 5.0, [11,1] := 0.7, [11,2] := 400.0, [11,3] := 75.0, [11,4] := 5.0, [11,5] := 800.0, [11,6] := 51.0, [11,8] := 100.0, [11,9] := 200.0, [11,14] := 7.5, [11,15] := 10.0, [12,0] := 5.0, [12,1] := 0.7, [12,2] := 400.0, [12,3] := 75.0, [12,4] := 5.0, [12,5] := 800.0, [12,6] := 51.0, [12,8] := 100.0, [12,9] := 200.0, [12,14] := 7.5, [12,15] := 10.0, [13,0] := 5.0, [13,1] := 0.7, [13,2] := 400.0, [13,3] := 75.0, [13,4] := 5.0, [13,5] := 800.0, [13,6] := 51.0, [13,8] := 100.0, [13,9] := 200.0, [13,14] := 7.5, [13,15] := 10.0, [14,0] := 5.0, [14,1] := 0.7, [14,2] := 400.0, [14,3] := 75.0, [14,4] := 5.0, [14,5] := 800.0, [14,6] := 51.0, [14,8] := 100.0, [14,9] := 200.0, [14,14] := 7.5, [14,15] := 10.0, [15,0] := 5.0, [15,1] := 0.7, [15,2] := 400.0, [15,3] := 75.0, [15,4] := 5.0, [15,5] := 800.0, [15,6] := 51.0, [15,8] := 100.0, [15,9] := 200.0, [15,14] := 7.5, [15,15] := 10.0, [16,0] := 5.0, [16,1] := 0.7, [16,2] := 400.0,
        [16,3] := 75.0, [16,4] := 5.0, [16,5] := 800.0, [16,6] := 51.0, [16,8] := 100.0, [16,9] := 200.0, [16,14] := 7.5, [16,15] := 10.0, [17,0] := 5.0, [17,1] := 0.7, [17,2] := 400.0, [17,3] := 75.0, [17,4] := 5.0, [17,5] := 800.0, [17,6] := 51.0, [17,8] := 100.0, [17,9] := 200.0, [17,14] := 7.5, [17,15] := 10.0, [18,0] := 5.0, [18,1] := 0.7, [18,2] := 400.0, [18,3] := 75.0, [18,4] := 5.0, [18,5] := 800.0, [18,6] := 51.0, [18,8] := 100.0, [18,9] := 200.0, [18,14] := 7.5, [18,15] := 10.0, [19,0] := 5.0, [19,1] := 0.7, [19,2] := 400.0, [19,3] := 75.0, [19,4] := 5.0, [19,5] := 800.0, [19,6] := 51.0, [19,8] := 100.0, [19,9] := 200.0, [19,14] := 7.5, [19,15] := 10.0, [20,0] := 5.0, [20,1] := 0.7, [20,2] := 400.0, [20,3] := 75.0, [20,4] := 5.0, [20,5] := 800.0, [20,6] := 51.0, [20,8] := 100.0, [20,9] := 200.0, [20,14] := 7.5, [20,15] := 10.0, [21,0] := 5.0, [21,1] := 0.7, [21,2] := 400.0, [21,3] := 75.0, [21,4] := 5.0, [21,5] := 800.0, [21,6] := 51.0, [21,8] := 100.0,
        [21,9] := 200.0, [21,14] := 7.5, [21,15] := 10.0, [22,0] := 5.0, [22,1] := 0.7, [22,2] := 400.0, [22,3] := 75.0, [22,4] := 5.0, [22,5] := 800.0, [22,6] := 51.0, [22,8] := 100.0, [22,9] := 200.0, [22,14] := 7.5, [22,15] := 10.0);
        [0,0]   // Filler A Deposit Stroke Distance
        [0,14]   // Flighted Conveyor Pan Release Min Position
        [0,15]   // Flighted Conveyor Pan Release Max Position
        [0,1]   // Filler A Deposit 1 Position
        [0,2]   // Filler A Deposit 2 Position
        [0,3]   // Filler A Deposit 3 Position
        [0,4]   // Blow-off Time
        [0,5]   // Blow-off Delay
        [0,6]   // Filler B Deposit Stroke Distance
        [0,7]   // Filler B Deposit 1 Position
        [0,8]   // Filler B Deposit 2 Position
        [0,9]   // Filler B Deposit 3 Position
   Recipe_Setpoints_REAL_Temp : REAL[20] := ([0] := 15.0, [1] := 0.7, [2] := 5.0, [3] := 500.0, [4] := 5.0, [5] := 1500.0, [6] := 500.0, [8] := 0.25, [9] := 200.0, [14] := 7.5, [15] := 10.0);
   Release_Bridge_Distance : REAL[10] := ([1] := -3.8, [2] := -7.65, [3] := -11.7);
   Release_MAG_Distance : REAL[10] := ([1] := -3.86, [2] := -7.65, [3] := -11.8);
   Releases_Dive : BOOL;
   Return_Speeds : DINT[10] := ([0] := 3, [1] := 7, [2] := 20, [3] := 30, [4] := 60);
   Sequencer_Auto : Sequencer_R2a := (Timer[0].PRE := 5, Timer[1].PRE := 50, Timer[10].PRE := 5, Timer[20].PRE := 200, Timer[30].PRE := 250, Timer[40].PRE := 50, Timer[50].PRE := 5, Timer[60].PRE := 5, Timer[70].PRE := 5, Timer[80].PRE := 5, Timer[90].PRE := 5);
   Sequencer_Home : Sequencer_R2a := (Timer[0].PRE := 5, Timer[1].PRE := 5, Timer[10].PRE := 1000, Timer[20].PRE := 5, Timer[30].PRE := 250, Timer[40].PRE := 5, Timer[50].PRE := 5, Timer[60].PRE := 250, Timer[70].PRE := 5, Timer[80].PRE := 500);
   Servo_Bridge_Shift : AXIS_CIP_DRIVE;
   Servo_Group_1 : MOTION_GROUP;   // Servo Bridge
   Servo_MC_Bridge_Shift : Axis_MC_R3b := (Direction_Rev_DINT := 1, Multiplier_Distance := -1.0, Multiplier_Speed := 0.5, Distance_Home_Offset := 2.0, Speed_Homing := 5.0, Speed_Jog_FWD := 10.0, Speed_Jog_REV := 10.0, Speed_Auto_REV := 8.0, Accel_Homing := 50.0, Accel_Jog := 20.0, Accel_Auto := 200.0, Decel_Estop := 100.0, Decel_Homing := 100.0, Decel_Jog := 50.0, Decel_Auto := 200.0, Status_Stopped := 1, Status_Safe_to_Move := 1, Timer_Jog_FWD_Delay.PRE := 250, Timer_Jog_REV_Delay.PRE := 250, Timer_Servo_Safe_to_Move.PRE := 5, Timer_Servo_Safe_to_Move.ACC := 5, Timer_Servo_Safe_to_Move.EN := 1, Timer_Servo_Safe_to_Move.DN := 1, OS[0] := 262, MSO.FLAGS := 570425344, MSO.DN := 1, MSO.STATE := 1, MSF.FLAGS := 33554432, MASR.FLAGS := 570425344, MASR.DN := 1, MASR.STATE := 1, MAFR.FLAGS := 570425344, MAFR.DN := 1, MAFR.STATE := 1, MAJ[0].FLAGS := 33554432, MAJ[1].FLAGS := 33554432, MAJ[2].FLAGS := 33554432, MAJ[3].FLAGS := 570425344, MAJ[3].DN := 1, MAJ_SPEED[0] := 5.0, MAJ_SPEED[1] := 5.0, MAJ_SPEED[2] := 2.5, MAJ_SPEED[3] := 2.5, MAJ_ACC[0] := 20.0, MAJ_ACC[1] := 20.0, MAJ_ACC[2] := 50.0, MAJ_ACC[3] := 50.0, MAJ_DEC[0] := 50.0, MAJ_DEC[1] := 50.0, MAJ_DEC[2] := 100.0, MAJ_DEC[3] := 100.0, MAM[0].FLAGS := 704643072, MAM[0].DN := 1, MAM[0].PC := 1, MAM[1].FLAGS := 704643072, MAM[1].DN := 1, MAM[1].PC := 1, MAM[2].FLAGS := 33554432, MAM_DISTANCE[0] := -2.0, MAM_DISTANCE[2] := -4.0,
        MAM_SPEED[0] := 2.5, MAM_SPEED[1] := 5.0, MAM_SPEED[2] := 50.0, MAM_ACC[0] := 50.0, MAM_ACC[1] := 200.0, MAM_ACC[2] := 150.0, MAM_DEC[0] := 100.0, MAM_DEC[1] := 200.0, MAM_DEC[2] := 150.0, MAS[0].FLAGS := 570425344, MAS[0].DN := 1, MAS[1].FLAGS := 33554432, MAS[2].FLAGS := 301989888, MAS[2].ER := 1, MAS[2].ERR := 78, MAS[3].FLAGS := 704643072, MAS[3].DN := 1, MAS[3].PC := 1, MAS_DEC[0] := 100.0, MAS_DEC[1] := 50.0, MAS_DEC[2] := 100.0, MAS_DEC[3] := 200.0, MAH[0].FLAGS := 704643072, MAH[0].DN := 1, MAH[0].PC := 1, MAH[0].STATE := 17, MAG[0].FLAGS := 570425344, MAG[0].DN := 1, MAG_DIRECTION[0] := 1, MAG_ACC[0] := 200.0, MAG_RATIO[0] := 10.0);
        .TIMER_TEST   // Test timer
   System : System_R2e := (HMI_Current_Screen := 1, HMI_PB_Auto := 1, HMI_PB_Clean := 1, HMI_Visible_Home_Servos := 1, Estop_Reset_Enabled := 1, Timer_Starting.PRE := 3000, Timer_Stopping.PRE := 3000, Timer_Stopping.ACC := 3000, Timer_EStop_Reset.PRE := 2000, Timer_EStop_Reset.ACC := 2000, Timer_EStop_Reset.EN := 1, Timer_EStop_Reset.DN := 1, Timer_Estop_OK.PRE := 3000, Timer_Estop_OK.ACC := 3000, Timer_Estop_OK.EN := 1, Timer_Estop_OK.DN := 1, Timer_Power_Up.PRE := 30000, Timer_Power_Up.ACC := 30000, Timer_Power_Up.EN := 1, Timer_Power_Up.DN := 1, Timer_Alarm_Timeout.PRE := 30000, Timer_Flasher_Slow_On.PRE := 400, Timer_Flasher_Slow_On.ACC := 201, Timer_Flasher_Slow_On.EN := 1, Timer_Flasher_Slow_On.TT := 1, Timer_Flasher_Slow_Off.PRE := 400, Timer_Flasher_Fast_On.PRE := 150, Timer_Flasher_Fast_On.ACC := 150, Timer_Flasher_Fast_On.EN := 1, Timer_Flasher_Fast_On.DN := 1, Timer_Flasher_Fast_Off.PRE := 150, Timer_Flasher_Fast_Off.ACC := 6, Timer_Flasher_Fast_Off.EN := 1, Timer_Flasher_Fast_Off.TT := 1, Timer_Servos_Home.PRE := 1000, Timer_Servos_Home.ACC := 1000, Timer_Servos_Home.EN := 1, Timer_Servos_Home.DN := 1, Timer_Alarm_Horn.PRE := 6000, Timer_Wipe_Screen.PRE := 10000, Mode_Auto := 1, Mode_Clean := 1, Mode_Integer := 3, Status_Estop_OK := 1, Status_DINT := 5, Servos_Homed := 1);
        .Mode_Prime   // System in Prime Mode
        .Mode_Auto   // System in Auto Mode
        .Timer_Flasher_Fast_On   // System Fast Flasher Timer On
        .Timer_Starting   // System Starting Timer
        .Timer_Starting.TT   // System Starting Timer Timing
        .Timer_Stopping   // System Stopping Timer
        .Timer_Stopping.EN   // System Stopping Timer Enabled
        .Timer_Stopping.DN   // System Stopping Timer Done
        .Timer_Flasher_Fast_Off   // System Fast Flasher Timer Off
        .Timer_Power_Up   // System Power Up Timer
        .Timer_Flasher_Slow_Off   // System Slow Flasher Timer Off
        .Status_Alarm   // Machine Alarm Active
        .Mode_Off   // System in Off Mode
        .Servos_OK   // System Servos OK
        .Timer_Flasher_Slow_On   // System Slow Flasher Timer On
        .Mode_Integer   // System Mode 0 = Prime 1 = Off 2 = Auto 3 = Clean
        .Timer_Estop_OK   // E-Stop OK Timer
   Test_Bits : BOOL[32];
   Timers : TIMER[20] := ([0].PRE := 5000, [1].PRE := 840, [2].PRE := 50, [2].ACC := 50, [2].EN := 1, [2].DN := 1, [3].PRE := 50, [3].ACC := 50, [3].EN := 1, [3].DN := 1, [4].PRE := 1000);   // x
        [4]   // TEST TIMER
        [0]   // Test Timer 0
        [1]   // TEST TIMER
        [3]   // MV Stopping
        [2]   // MV_Moving
   Trigger_Counter : COUNTER := (PRE := 3, ACC := 2);
   trigger_Denester : BOOL;
   Ulma_Running_Bypass : BOOL := 1;
   USE_ENCODER : BOOL;
END_VAR

PROGRAM MainProgram   (* main routine File_001_Main *)

ROUTINE File_001_Main   (* ladder *)
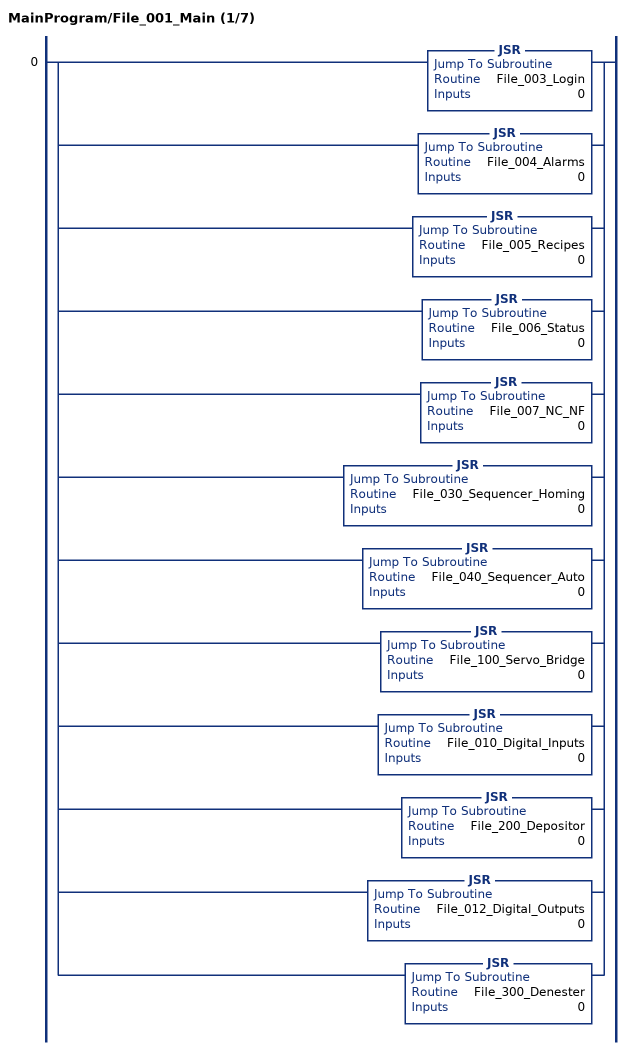
   0: [JSR(File_003_Login,0) ,JSR(File_004_Alarms,0) ,JSR(File_005_Recipes,0) ,JSR(File_006_Status,0) ,JSR(File_007_NC_NF,0) ,JSR(File_030_Sequencer_Homing,0) ,JSR(File_040_Sequencer_Auto,0) ,JSR(File_100_Servo_Bridge,0) ,JSR(File_010_Digital_Inputs,0) ,JSR(File_200_Depositor,0) ,JSR(File_012_Digital_Outputs,0) ,JSR(File_300_Denester,0) ];
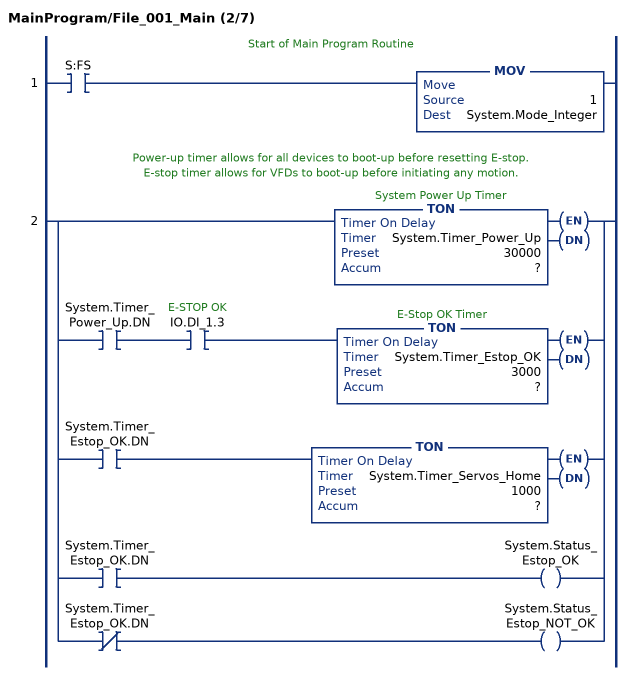
   // Start of Main Program Routine
   1: XIC(S:FS)MOV(1,System.Mode_Integer);
   // Power-up timer allows for all devices to boot-up before resetting E-stop.
   // E-stop timer allows for VFDs to boot-up before initiating any motion.
   2: [TON(System.Timer_Power_Up,?,?) ,XIC(System.Timer_Power_Up.DN) XIC(IO.DI_1.3) TON(System.Timer_Estop_OK,?,?) ,XIC(System.Timer_Estop_OK.DN) TON(System.Timer_Servos_Home,?,?) ,XIC(System.Timer_Estop_OK.DN) OTE(System.Status_Estop_OK) ,XIO(System.Timer_Estop_OK.DN) OTE(System.Status_Estop_NOT_OK) ];
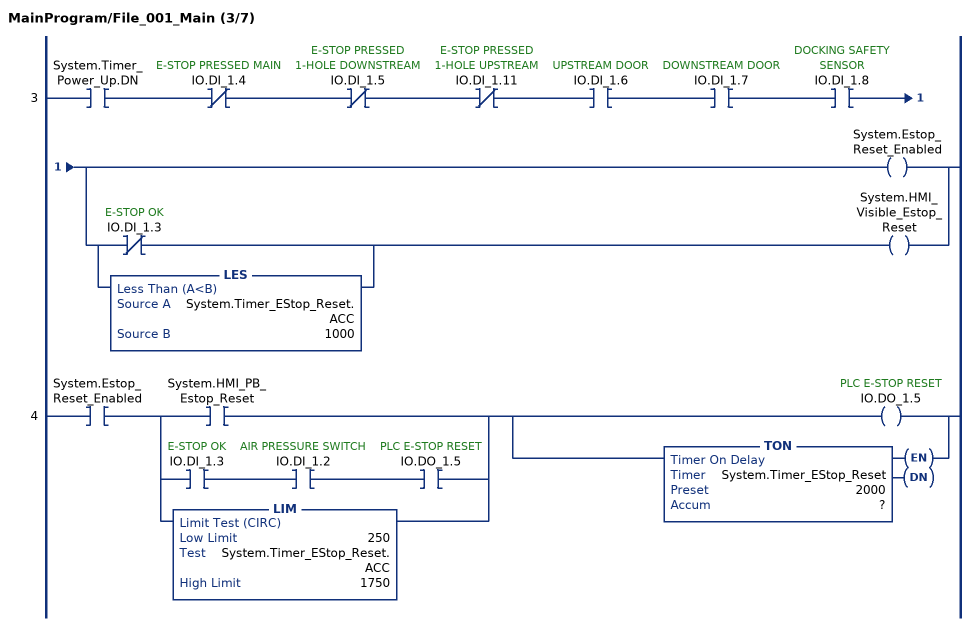
   3: XIC(System.Timer_Power_Up.DN)XIO(IO.DI_1.4)XIO(IO.DI_1.5)XIO(IO.DI_1.11)XIC(IO.DI_1.6)XIC(IO.DI_1.7)XIC(IO.DI_1.8)[OTE(System.Estop_Reset_Enabled) ,[XIO(IO.DI_1.3) ,LES(System.Timer_EStop_Reset.ACC,1000) ] OTE(System.HMI_Visible_Estop_Reset) ];
   4: XIC(System.Estop_Reset_Enabled)[XIC(System.HMI_PB_Estop_Reset) ,XIC(IO.DI_1.3) XIC(IO.DI_1.2) XIC(IO.DO_1.5) ,LIM(250,System.Timer_EStop_Reset.ACC,1750) ][OTE(IO.DO_1.5) ,TON(System.Timer_EStop_Reset,?,?) ];
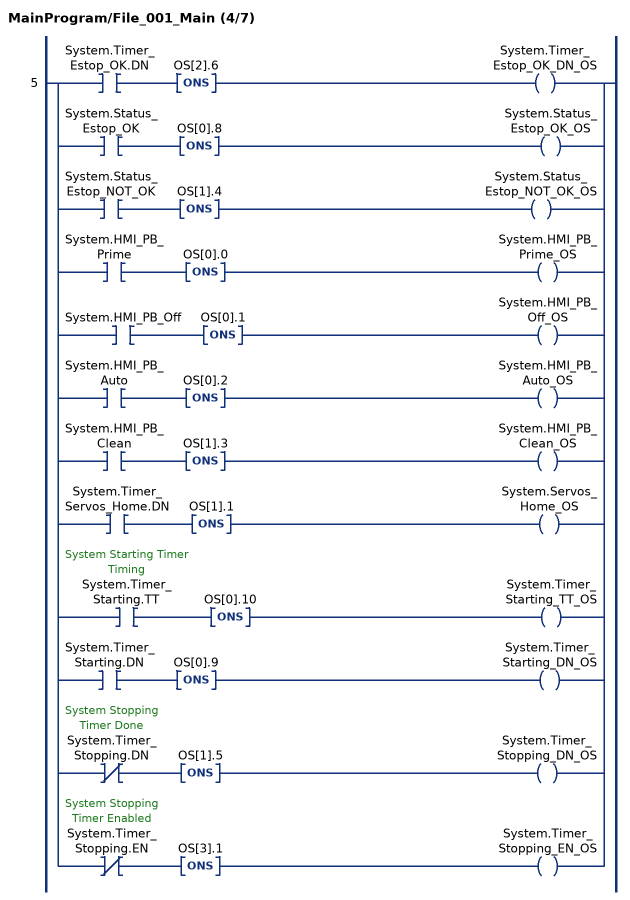
   5: [XIC(System.Timer_Estop_OK.DN) ONS(OS[2].6) OTE(System.Timer_Estop_OK_DN_OS) ,XIC(System.Status_Estop_OK) ONS(OS[0].8) OTE(System.Status_Estop_OK_OS) ,XIC(System.Status_Estop_NOT_OK) ONS(OS[1].4) OTE(System.Status_Estop_NOT_OK_OS) ,XIC(System.HMI_PB_Prime) ONS(OS[0].0) OTE(System.HMI_PB_Prime_OS) ,XIC(System.HMI_PB_Off) ONS(OS[0].1) OTE(System.HMI_PB_Off_OS) ,XIC(System.HMI_PB_Auto) ONS(OS[0].2) OTE(System.HMI_PB_Auto_OS) ,XIC(System.HMI_PB_Clean) ONS(OS[1].3) OTE(System.HMI_PB_Clean_OS) ,XIC(System.Timer_Servos_Home.DN) ONS(OS[1].1) OTE(System.Servos_Home_OS) ,XIC(System.Timer_Starting.TT) ONS(OS[0].10) OTE(System.Timer_Starting_TT_OS) ,XIC(System.Timer_Starting.DN) ONS(OS[0].9) OTE(System.Timer_Starting_DN_OS) ,XIO(System.Timer_Stopping.DN) ONS(OS[1].5) OTE(System.Timer_Stopping_DN_OS) ,XIO(System.Timer_Stopping.EN) ONS(OS[3].1) OTE(System.Timer_Stopping_EN_OS) ];
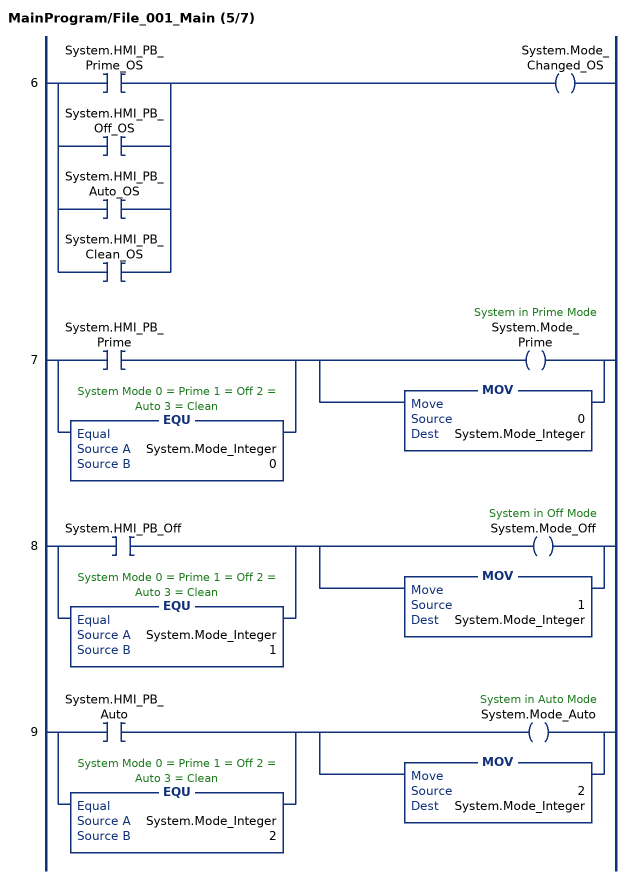
   6: [XIC(System.HMI_PB_Prime_OS) ,XIC(System.HMI_PB_Off_OS) ,XIC(System.HMI_PB_Auto_OS) ,XIC(System.HMI_PB_Clean_OS) ]OTE(System.Mode_Changed_OS);
   7: [XIC(System.HMI_PB_Prime) ,EQU(System.Mode_Integer,0) ][OTE(System.Mode_Prime) ,MOV(0,System.Mode_Integer) ];
   8: [XIC(System.HMI_PB_Off) ,EQU(System.Mode_Integer,1) ][OTE(System.Mode_Off) ,MOV(1,System.Mode_Integer) ];
   9: [XIC(System.HMI_PB_Auto) ,EQU(System.Mode_Integer,2) ][OTE(System.Mode_Auto) ,MOV(2,System.Mode_Integer) ];
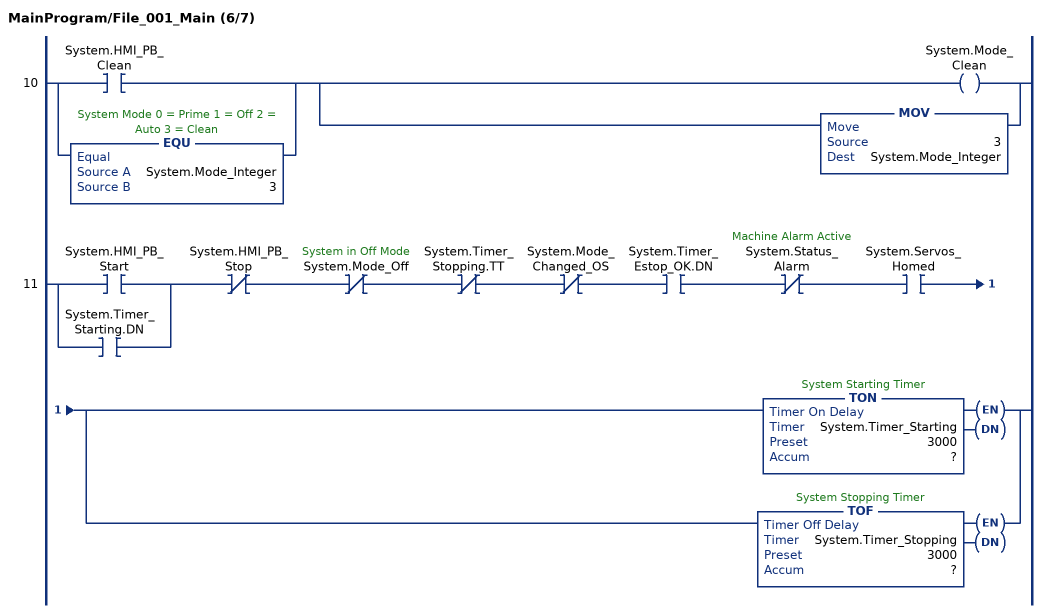
   10: [XIC(System.HMI_PB_Clean) ,EQU(System.Mode_Integer,3) ][OTE(System.Mode_Clean) ,MOV(3,System.Mode_Integer) ];
   11: [XIC(System.HMI_PB_Start) ,XIC(System.Timer_Starting.DN) ]XIO(System.HMI_PB_Stop)XIO(System.Mode_Off)XIO(System.Timer_Stopping.TT)XIO(System.Mode_Changed_OS)XIC(System.Timer_Estop_OK.DN)XIO(System.Status_Alarm)XIC(System.Servos_Homed)[TON(System.Timer_Starting,?,?) ,TOF(System.Timer_Stopping,?,?) ];
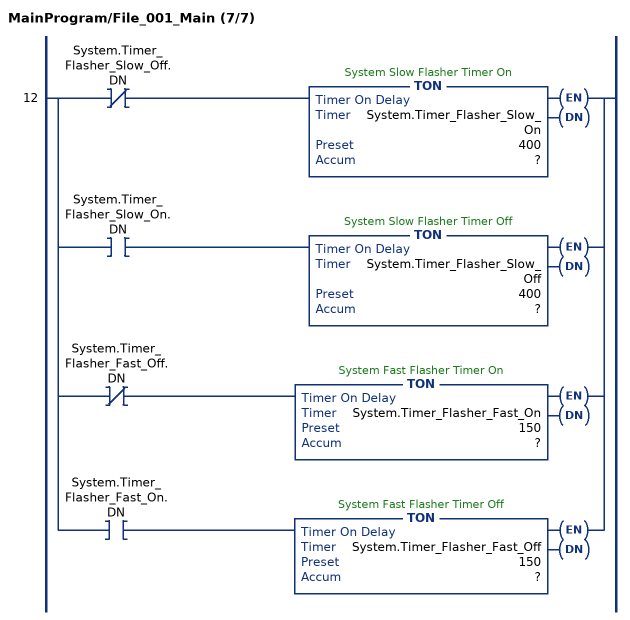
   12: [[XIO(System.Timer_Flasher_Slow_Off.DN) TON(System.Timer_Flasher_Slow_On,?,?) ,XIC(System.Timer_Flasher_Slow_On.DN) TON(System.Timer_Flasher_Slow_Off,?,?) ] ,[XIO(System.Timer_Flasher_Fast_Off.DN) TON(System.Timer_Flasher_Fast_On,?,?) ,XIC(System.Timer_Flasher_Fast_On.DN) TON(System.Timer_Flasher_Fast_Off,?,?) ] ];
END_ROUTINE

ROUTINE File_003_Login   (* ladder *)
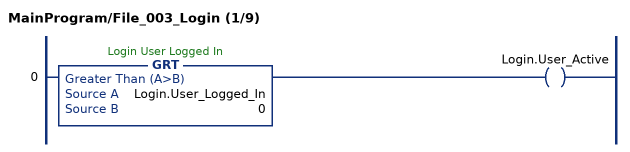
   0: GRT(Login.User_Logged_In,0)OTE(Login.User_Active);
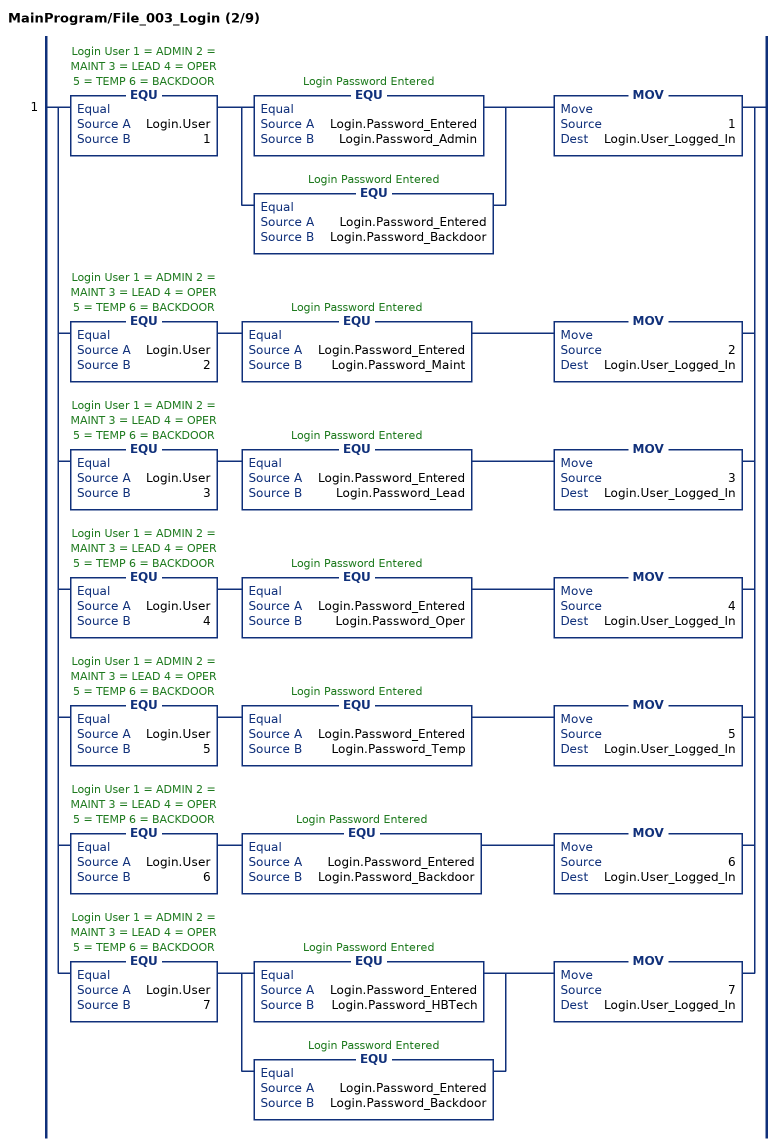
   1: [EQU(Login.User,1) [EQU(Login.Password_Entered,Login.Password_Admin) ,EQU(Login.Password_Entered,Login.Password_Backdoor) ] MOV(1,Login.User_Logged_In) ,EQU(Login.User,2) EQU(Login.Password_Entered,Login.Password_Maint) MOV(2,Login.User_Logged_In) ,EQU(Login.User,3) EQU(Login.Password_Entered,Login.Password_Lead) MOV(3,Login.User_Logged_In) ,EQU(Login.User,4) EQU(Login.Password_Entered,Login.Password_Oper) MOV(4,Login.User_Logged_In) ,EQU(Login.User,5) EQU(Login.Password_Entered,Login.Password_Temp) MOV(5,Login.User_Logged_In) ,EQU(Login.User,6) EQU(Login.Password_Entered,Login.Password_Backdoor) MOV(6,Login.User_Logged_In) ,EQU(Login.User,7) [EQU(Login.Password_Entered,Login.Password_HBTech) ,EQU(Login.Password_Entered,Login.Password_Backdoor) ] MOV(7,Login.User_Logged_In) ];
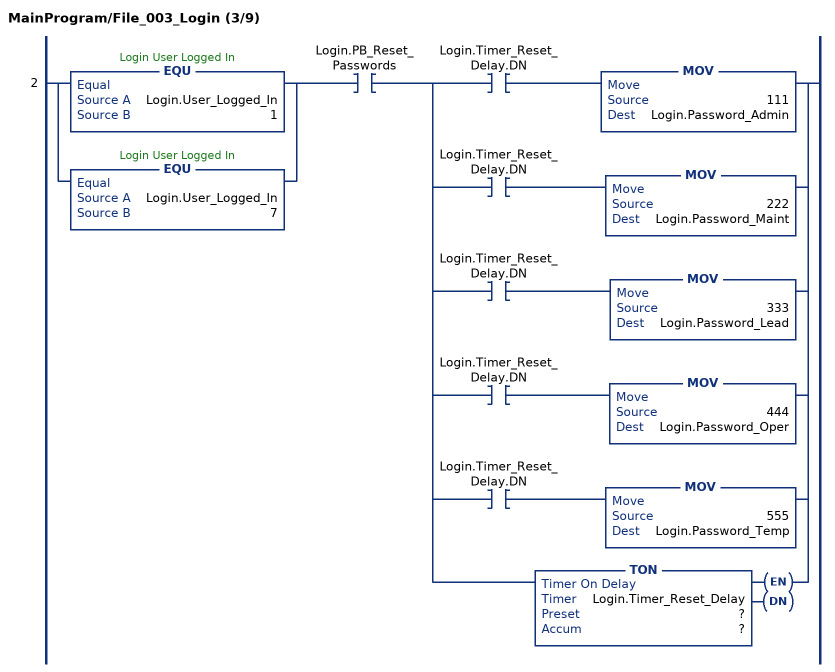
   2: [EQU(Login.User_Logged_In,1) ,EQU(Login.User_Logged_In,7) ]XIC(Login.PB_Reset_Passwords)[XIC(Login.Timer_Reset_Delay.DN) MOV(111,Login.Password_Admin) ,XIC(Login.Timer_Reset_Delay.DN) MOV(222,Login.Password_Maint) ,XIC(Login.Timer_Reset_Delay.DN) MOV(333,Login.Password_Lead) ,XIC(Login.Timer_Reset_Delay.DN) MOV(444,Login.Password_Oper) ,XIC(Login.Timer_Reset_Delay.DN) MOV(555,Login.Password_Temp) ,TON(Login.Timer_Reset_Delay,?,?) ];
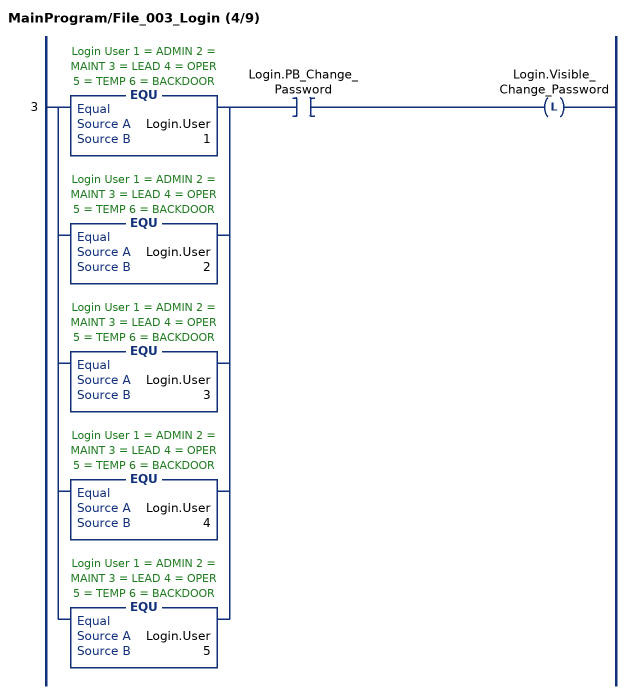
   3: [EQU(Login.User,1) ,EQU(Login.User,2) ,EQU(Login.User,3) ,EQU(Login.User,4) ,EQU(Login.User,5) ]XIC(Login.PB_Change_Password)OTL(Login.Visible_Change_Password);
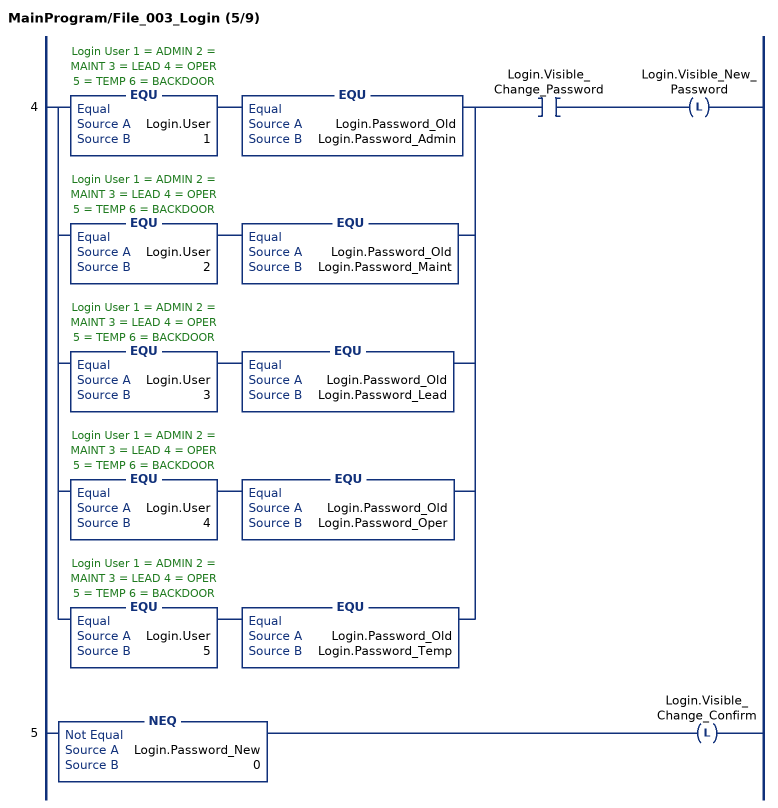
   4: [EQU(Login.User,1) EQU(Login.Password_Old,Login.Password_Admin) ,EQU(Login.User,2) EQU(Login.Password_Old,Login.Password_Maint) ,EQU(Login.User,3) EQU(Login.Password_Old,Login.Password_Lead) ,EQU(Login.User,4) EQU(Login.Password_Old,Login.Password_Oper) ,EQU(Login.User,5) EQU(Login.Password_Old,Login.Password_Temp) ]XIC(Login.Visible_Change_Password)OTL(Login.Visible_New_Password);
   5: NEQ(Login.Password_New,0)OTL(Login.Visible_Change_Confirm);
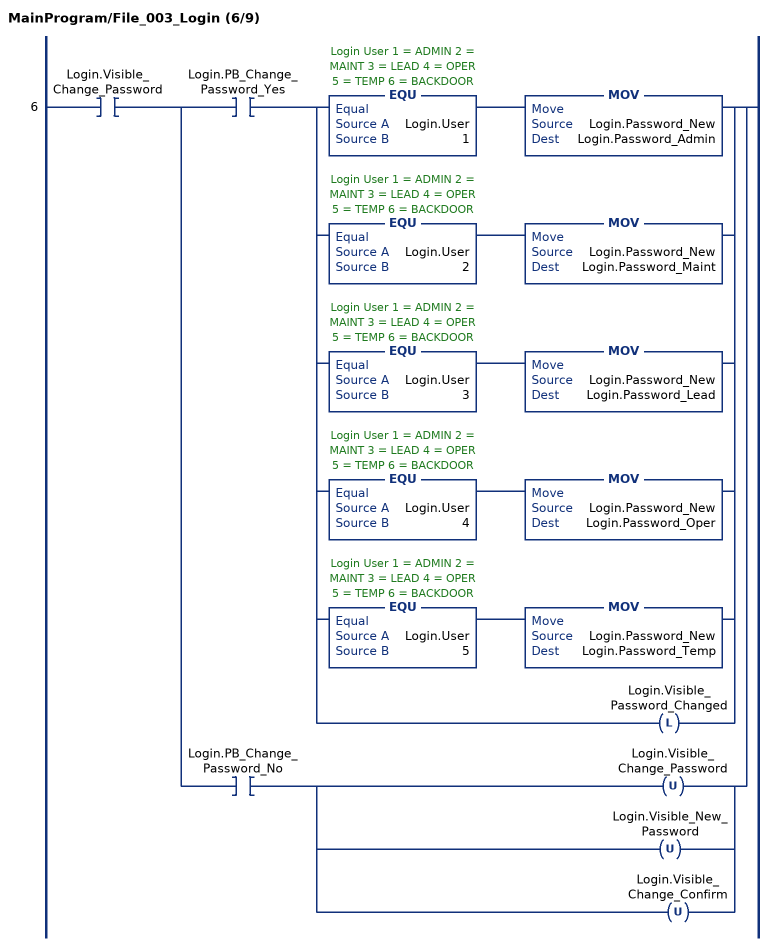
   6: XIC(Login.Visible_Change_Password)[XIC(Login.PB_Change_Password_Yes) [EQU(Login.User,1) MOV(Login.Password_New,Login.Password_Admin) ,EQU(Login.User,2) MOV(Login.Password_New,Login.Password_Maint) ,EQU(Login.User,3) MOV(Login.Password_New,Login.Password_Lead) ,EQU(Login.User,4) MOV(Login.Password_New,Login.Password_Oper) ,EQU(Login.User,5) MOV(Login.Password_New,Login.Password_Temp) ,OTL(Login.Visible_Password_Changed) ] ,XIC(Login.PB_Change_Password_No) [OTU(Login.Visible_Change_Password) ,OTU(Login.Visible_New_Password) ,OTU(Login.Visible_Change_Confirm) ] ];
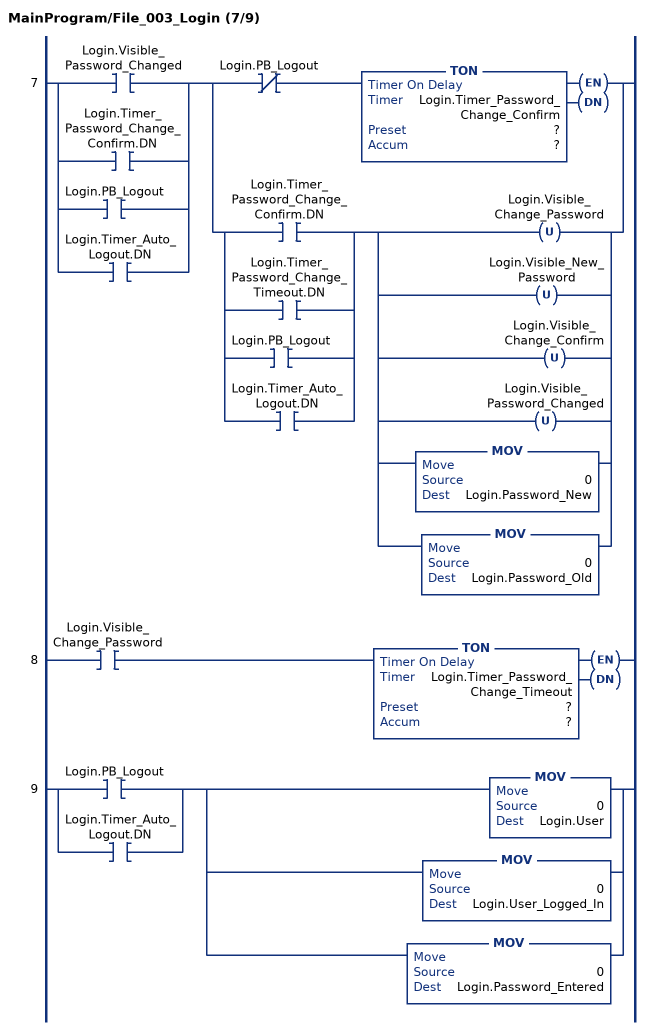
   7: [XIC(Login.Visible_Password_Changed) ,XIC(Login.Timer_Password_Change_Confirm.DN) ,XIC(Login.PB_Logout) ,XIC(Login.Timer_Auto_Logout.DN) ][XIO(Login.PB_Logout) TON(Login.Timer_Password_Change_Confirm,?,?) ,[XIC(Login.Timer_Password_Change_Confirm.DN) ,XIC(Login.Timer_Password_Change_Timeout.DN) ,XIC(Login.PB_Logout) ,XIC(Login.Timer_Auto_Logout.DN) ] [OTU(Login.Visible_Change_Password) ,OTU(Login.Visible_New_Password) ,OTU(Login.Visible_Change_Confirm) ,OTU(Login.Visible_Password_Changed) ,MOV(0,Login.Password_New) ,MOV(0,Login.Password_Old) ] ];
   8: XIC(Login.Visible_Change_Password)TON(Login.Timer_Password_Change_Timeout,?,?);
   9: [XIC(Login.PB_Logout) ,XIC(Login.Timer_Auto_Logout.DN) ][MOV(0,Login.User) ,MOV(0,Login.User_Logged_In) ,MOV(0,Login.Password_Entered) ];
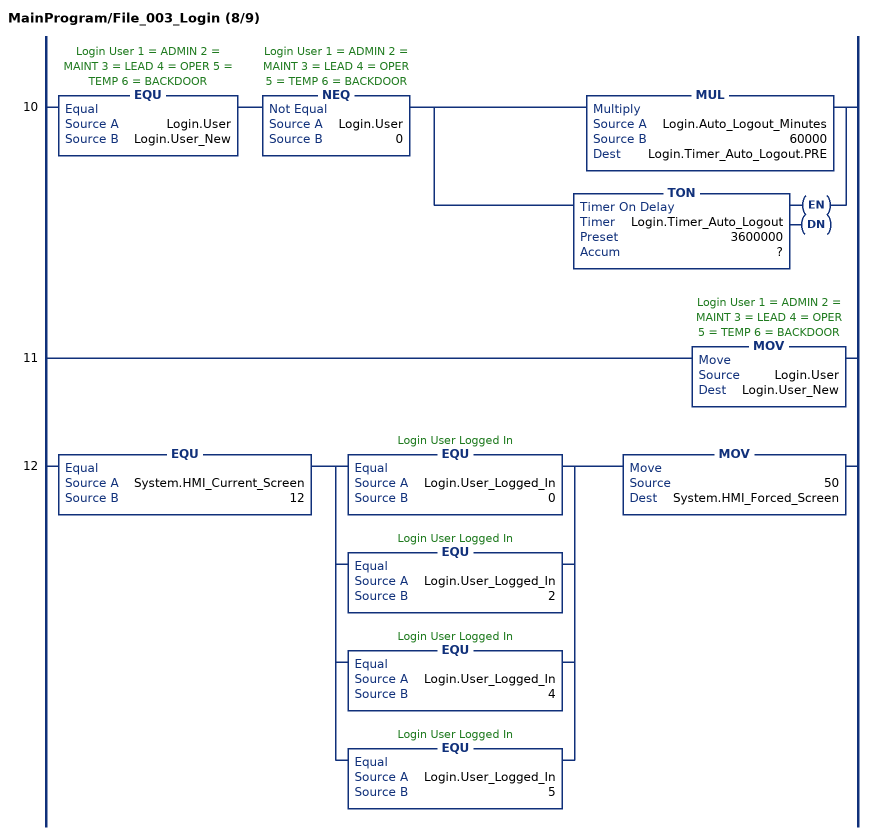
   10: EQU(Login.User,Login.User_New)NEQ(Login.User,0)[MUL(Login.Auto_Logout_Minutes,60000,Login.Timer_Auto_Logout.PRE) ,TON(Login.Timer_Auto_Logout,?,?) ];
   11: MOV(Login.User,Login.User_New);
   12: EQU(System.HMI_Current_Screen,12)[EQU(Login.User_Logged_In,0) ,EQU(Login.User_Logged_In,2) ,EQU(Login.User_Logged_In,4) ,EQU(Login.User_Logged_In,5) ]MOV(50,System.HMI_Forced_Screen);
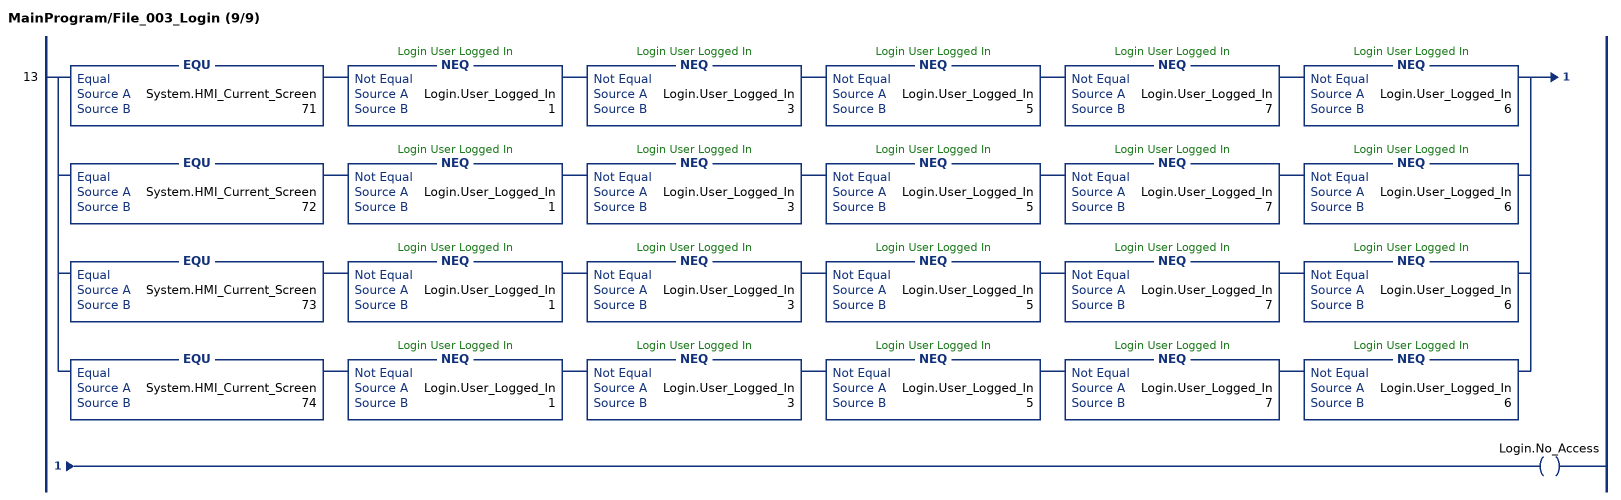
   13: [EQU(System.HMI_Current_Screen,71) NEQ(Login.User_Logged_In,1) NEQ(Login.User_Logged_In,3) NEQ(Login.User_Logged_In,5) NEQ(Login.User_Logged_In,7) NEQ(Login.User_Logged_In,6) ,EQU(System.HMI_Current_Screen,72) NEQ(Login.User_Logged_In,1) NEQ(Login.User_Logged_In,3) NEQ(Login.User_Logged_In,5) NEQ(Login.User_Logged_In,7) NEQ(Login.User_Logged_In,6) ,EQU(System.HMI_Current_Screen,73) NEQ(Login.User_Logged_In,1) NEQ(Login.User_Logged_In,3) NEQ(Login.User_Logged_In,5) NEQ(Login.User_Logged_In,7) NEQ(Login.User_Logged_In,6) ,EQU(System.HMI_Current_Screen,74) NEQ(Login.User_Logged_In,1) NEQ(Login.User_Logged_In,3) NEQ(Login.User_Logged_In,5) NEQ(Login.User_Logged_In,7) NEQ(Login.User_Logged_In,6) ]OTE(Login.No_Access);
END_ROUTINE

ROUTINE File_004_Alarms   (* ladder *)
// Alarms to HMI
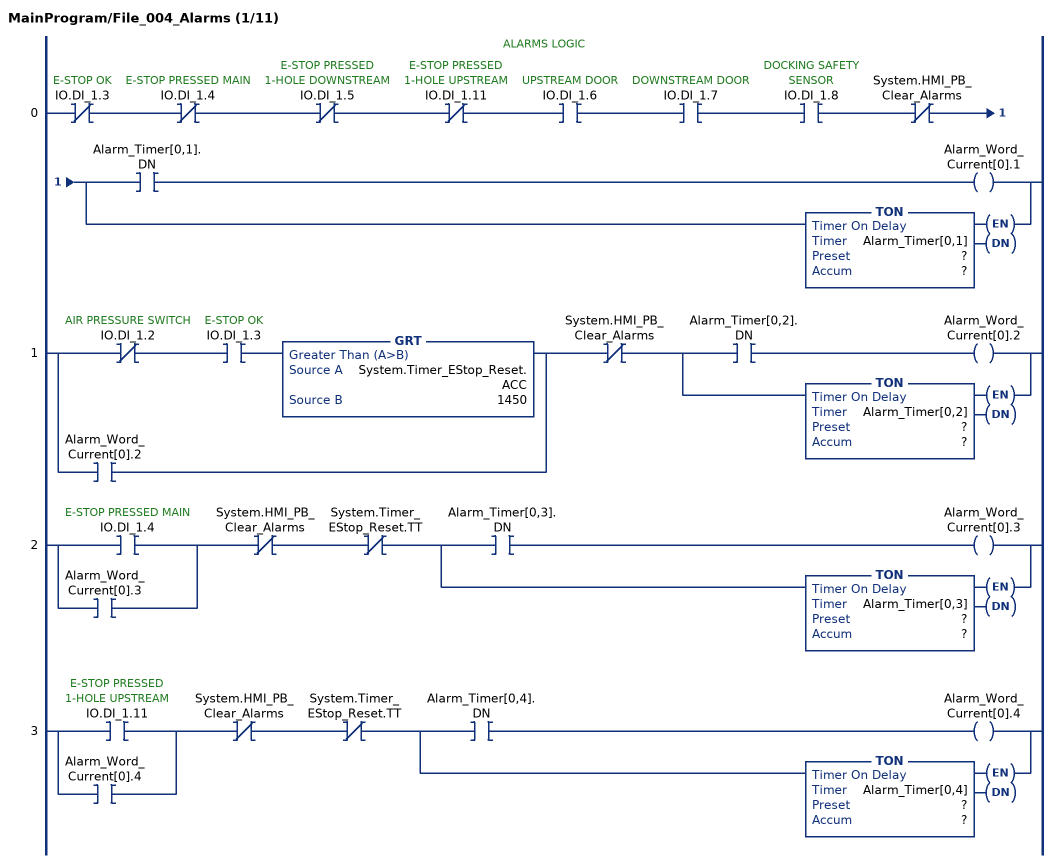
   // ALARMS LOGIC
   0: XIO(IO.DI_1.3)XIO(IO.DI_1.4)XIO(IO.DI_1.5)XIO(IO.DI_1.11)XIC(IO.DI_1.6)XIC(IO.DI_1.7)XIC(IO.DI_1.8)XIO(System.HMI_PB_Clear_Alarms)[XIC(Alarm_Timer[0,1].DN) OTE(Alarm_Word_Current[0].1) ,TON(Alarm_Timer[0,1],?,?) ];
   1: [XIO(IO.DI_1.2) XIC(IO.DI_1.3) GRT(System.Timer_EStop_Reset.ACC,1450) ,XIC(Alarm_Word_Current[0].2) ]XIO(System.HMI_PB_Clear_Alarms)[XIC(Alarm_Timer[0,2].DN) OTE(Alarm_Word_Current[0].2) ,TON(Alarm_Timer[0,2],?,?) ];
   2: [XIC(IO.DI_1.4) ,XIC(Alarm_Word_Current[0].3) ]XIO(System.HMI_PB_Clear_Alarms)XIO(System.Timer_EStop_Reset.TT)[XIC(Alarm_Timer[0,3].DN) OTE(Alarm_Word_Current[0].3) ,TON(Alarm_Timer[0,3],?,?) ];
   3: [XIC(IO.DI_1.11) ,XIC(Alarm_Word_Current[0].4) ]XIO(System.HMI_PB_Clear_Alarms)XIO(System.Timer_EStop_Reset.TT)[XIC(Alarm_Timer[0,4].DN) OTE(Alarm_Word_Current[0].4) ,TON(Alarm_Timer[0,4],?,?) ];
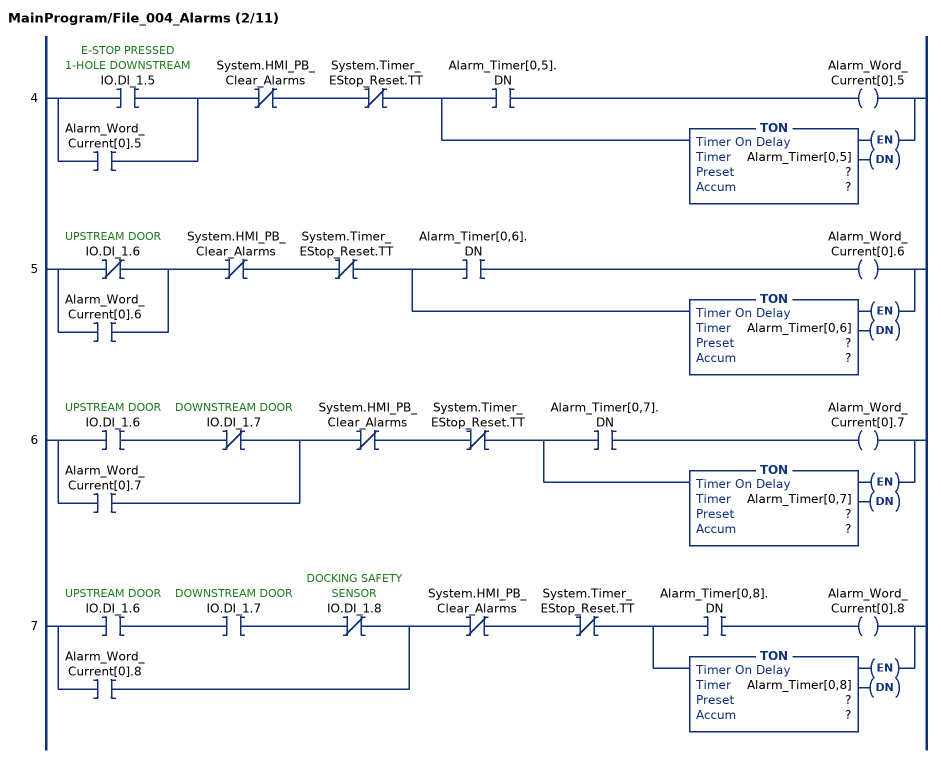
   4: [XIC(IO.DI_1.5) ,XIC(Alarm_Word_Current[0].5) ]XIO(System.HMI_PB_Clear_Alarms)XIO(System.Timer_EStop_Reset.TT)[XIC(Alarm_Timer[0,5].DN) OTE(Alarm_Word_Current[0].5) ,TON(Alarm_Timer[0,5],?,?) ];
   5: [XIO(IO.DI_1.6) ,XIC(Alarm_Word_Current[0].6) ]XIO(System.HMI_PB_Clear_Alarms)XIO(System.Timer_EStop_Reset.TT)[XIC(Alarm_Timer[0,6].DN) OTE(Alarm_Word_Current[0].6) ,TON(Alarm_Timer[0,6],?,?) ];
   6: [XIC(IO.DI_1.6) XIO(IO.DI_1.7) ,XIC(Alarm_Word_Current[0].7) ]XIO(System.HMI_PB_Clear_Alarms)XIO(System.Timer_EStop_Reset.TT)[XIC(Alarm_Timer[0,7].DN) OTE(Alarm_Word_Current[0].7) ,TON(Alarm_Timer[0,7],?,?) ];
   7: [XIC(IO.DI_1.6) XIC(IO.DI_1.7) XIO(IO.DI_1.8) ,XIC(Alarm_Word_Current[0].8) ]XIO(System.HMI_PB_Clear_Alarms)XIO(System.Timer_EStop_Reset.TT)[XIC(Alarm_Timer[0,8].DN) OTE(Alarm_Word_Current[0].8) ,TON(Alarm_Timer[0,8],?,?) ];
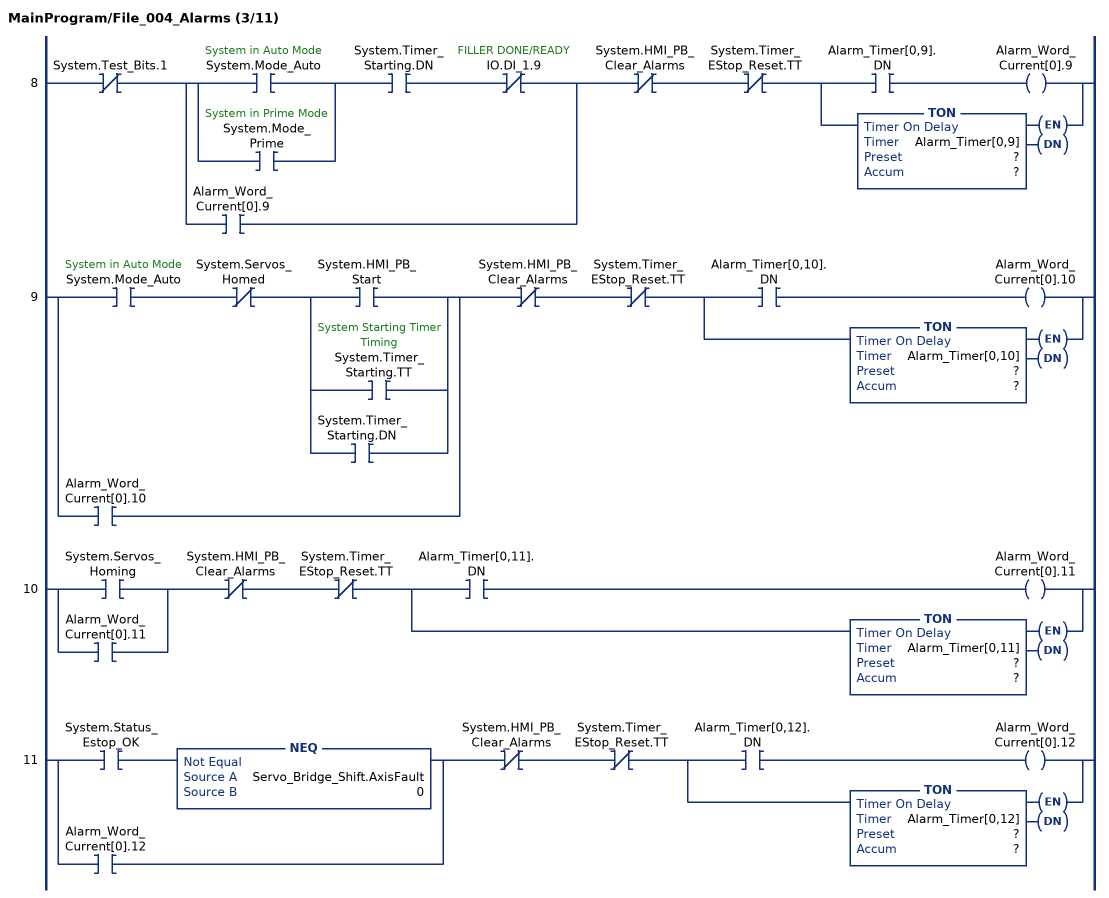
   8: XIO(System.Test_Bits.1)[[XIC(System.Mode_Auto) ,XIC(System.Mode_Prime) ] XIC(System.Timer_Starting.DN) XIO(IO.DI_1.9) ,XIC(Alarm_Word_Current[0].9) ]XIO(System.HMI_PB_Clear_Alarms)XIO(System.Timer_EStop_Reset.TT)[XIC(Alarm_Timer[0,9].DN) OTE(Alarm_Word_Current[0].9) ,TON(Alarm_Timer[0,9],?,?) ];
   9: [XIC(System.Mode_Auto) XIO(System.Servos_Homed) [XIC(System.HMI_PB_Start) ,XIC(System.Timer_Starting.TT) ,XIC(System.Timer_Starting.DN) ] ,XIC(Alarm_Word_Current[0].10) ]XIO(System.HMI_PB_Clear_Alarms)XIO(System.Timer_EStop_Reset.TT)[XIC(Alarm_Timer[0,10].DN) OTE(Alarm_Word_Current[0].10) ,TON(Alarm_Timer[0,10],?,?) ];
   10: [XIC(System.Servos_Homing) ,XIC(Alarm_Word_Current[0].11) ]XIO(System.HMI_PB_Clear_Alarms)XIO(System.Timer_EStop_Reset.TT)[XIC(Alarm_Timer[0,11].DN) OTE(Alarm_Word_Current[0].11) ,TON(Alarm_Timer[0,11],?,?) ];
   11: [XIC(System.Status_Estop_OK) NEQ(Servo_Bridge_Shift.AxisFault,0) ,XIC(Alarm_Word_Current[0].12) ]XIO(System.HMI_PB_Clear_Alarms)XIO(System.Timer_EStop_Reset.TT)[XIC(Alarm_Timer[0,12].DN) OTE(Alarm_Word_Current[0].12) ,TON(Alarm_Timer[0,12],?,?) ];
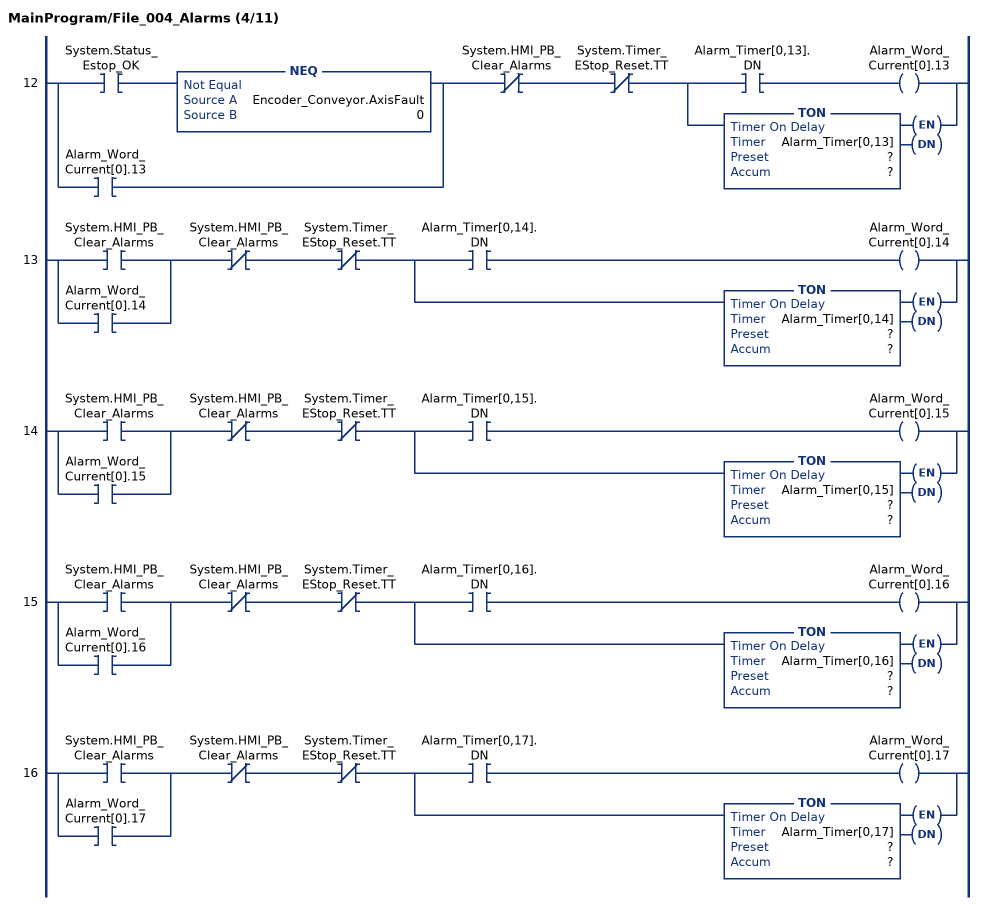
   12: [XIC(System.Status_Estop_OK) NEQ(Encoder_Conveyor.AxisFault,0) ,XIC(Alarm_Word_Current[0].13) ]XIO(System.HMI_PB_Clear_Alarms)XIO(System.Timer_EStop_Reset.TT)[XIC(Alarm_Timer[0,13].DN) OTE(Alarm_Word_Current[0].13) ,TON(Alarm_Timer[0,13],?,?) ];
   13: [XIC(System.HMI_PB_Clear_Alarms) ,XIC(Alarm_Word_Current[0].14) ]XIO(System.HMI_PB_Clear_Alarms)XIO(System.Timer_EStop_Reset.TT)[XIC(Alarm_Timer[0,14].DN) OTE(Alarm_Word_Current[0].14) ,TON(Alarm_Timer[0,14],?,?) ];
   14: [XIC(System.HMI_PB_Clear_Alarms) ,XIC(Alarm_Word_Current[0].15) ]XIO(System.HMI_PB_Clear_Alarms)XIO(System.Timer_EStop_Reset.TT)[XIC(Alarm_Timer[0,15].DN) OTE(Alarm_Word_Current[0].15) ,TON(Alarm_Timer[0,15],?,?) ];
   15: [XIC(System.HMI_PB_Clear_Alarms) ,XIC(Alarm_Word_Current[0].16) ]XIO(System.HMI_PB_Clear_Alarms)XIO(System.Timer_EStop_Reset.TT)[XIC(Alarm_Timer[0,16].DN) OTE(Alarm_Word_Current[0].16) ,TON(Alarm_Timer[0,16],?,?) ];
   16: [XIC(System.HMI_PB_Clear_Alarms) ,XIC(Alarm_Word_Current[0].17) ]XIO(System.HMI_PB_Clear_Alarms)XIO(System.Timer_EStop_Reset.TT)[XIC(Alarm_Timer[0,17].DN) OTE(Alarm_Word_Current[0].17) ,TON(Alarm_Timer[0,17],?,?) ];
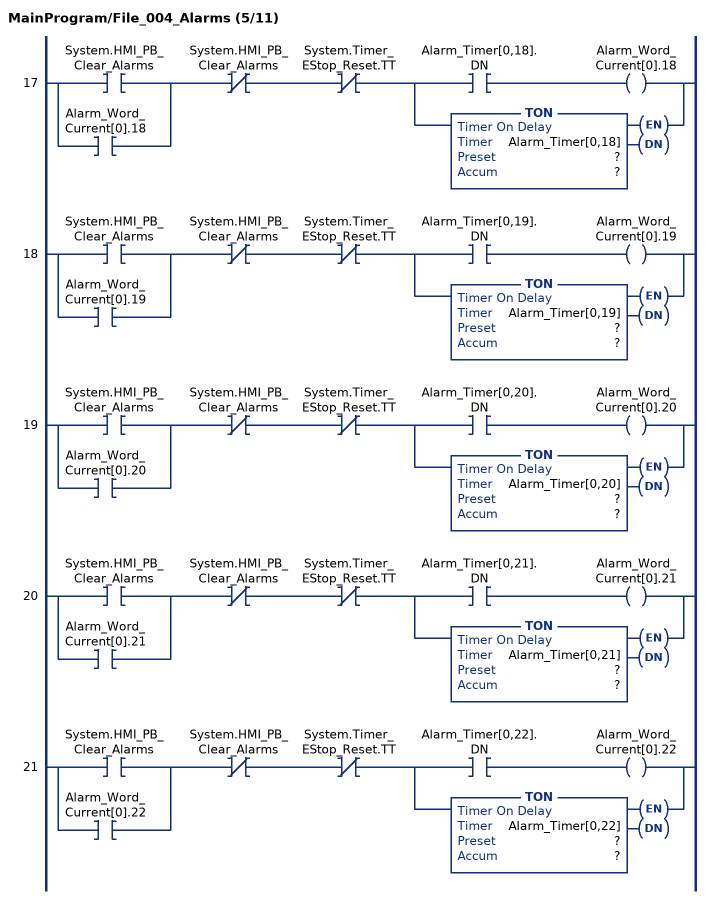
   17: [XIC(System.HMI_PB_Clear_Alarms) ,XIC(Alarm_Word_Current[0].18) ]XIO(System.HMI_PB_Clear_Alarms)XIO(System.Timer_EStop_Reset.TT)[XIC(Alarm_Timer[0,18].DN) OTE(Alarm_Word_Current[0].18) ,TON(Alarm_Timer[0,18],?,?) ];
   18: [XIC(System.HMI_PB_Clear_Alarms) ,XIC(Alarm_Word_Current[0].19) ]XIO(System.HMI_PB_Clear_Alarms)XIO(System.Timer_EStop_Reset.TT)[XIC(Alarm_Timer[0,19].DN) OTE(Alarm_Word_Current[0].19) ,TON(Alarm_Timer[0,19],?,?) ];
   19: [XIC(System.HMI_PB_Clear_Alarms) ,XIC(Alarm_Word_Current[0].20) ]XIO(System.HMI_PB_Clear_Alarms)XIO(System.Timer_EStop_Reset.TT)[XIC(Alarm_Timer[0,20].DN) OTE(Alarm_Word_Current[0].20) ,TON(Alarm_Timer[0,20],?,?) ];
   20: [XIC(System.HMI_PB_Clear_Alarms) ,XIC(Alarm_Word_Current[0].21) ]XIO(System.HMI_PB_Clear_Alarms)XIO(System.Timer_EStop_Reset.TT)[XIC(Alarm_Timer[0,21].DN) OTE(Alarm_Word_Current[0].21) ,TON(Alarm_Timer[0,21],?,?) ];
   21: [XIC(System.HMI_PB_Clear_Alarms) ,XIC(Alarm_Word_Current[0].22) ]XIO(System.HMI_PB_Clear_Alarms)XIO(System.Timer_EStop_Reset.TT)[XIC(Alarm_Timer[0,22].DN) OTE(Alarm_Word_Current[0].22) ,TON(Alarm_Timer[0,22],?,?) ];
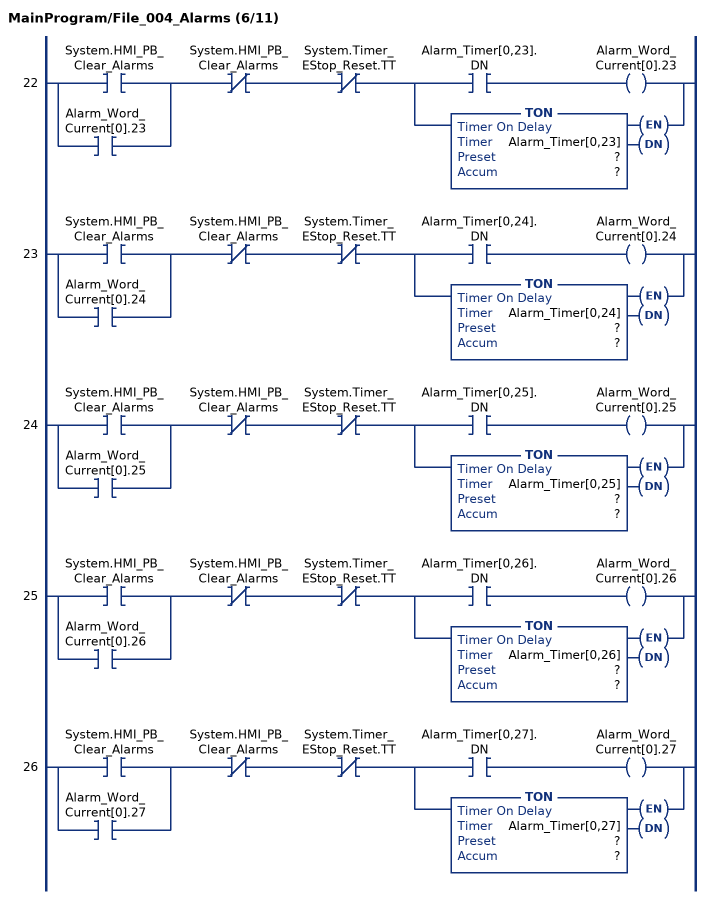
   22: [XIC(System.HMI_PB_Clear_Alarms) ,XIC(Alarm_Word_Current[0].23) ]XIO(System.HMI_PB_Clear_Alarms)XIO(System.Timer_EStop_Reset.TT)[XIC(Alarm_Timer[0,23].DN) OTE(Alarm_Word_Current[0].23) ,TON(Alarm_Timer[0,23],?,?) ];
   23: [XIC(System.HMI_PB_Clear_Alarms) ,XIC(Alarm_Word_Current[0].24) ]XIO(System.HMI_PB_Clear_Alarms)XIO(System.Timer_EStop_Reset.TT)[XIC(Alarm_Timer[0,24].DN) OTE(Alarm_Word_Current[0].24) ,TON(Alarm_Timer[0,24],?,?) ];
   24: [XIC(System.HMI_PB_Clear_Alarms) ,XIC(Alarm_Word_Current[0].25) ]XIO(System.HMI_PB_Clear_Alarms)XIO(System.Timer_EStop_Reset.TT)[XIC(Alarm_Timer[0,25].DN) OTE(Alarm_Word_Current[0].25) ,TON(Alarm_Timer[0,25],?,?) ];
   25: [XIC(System.HMI_PB_Clear_Alarms) ,XIC(Alarm_Word_Current[0].26) ]XIO(System.HMI_PB_Clear_Alarms)XIO(System.Timer_EStop_Reset.TT)[XIC(Alarm_Timer[0,26].DN) OTE(Alarm_Word_Current[0].26) ,TON(Alarm_Timer[0,26],?,?) ];
   26: [XIC(System.HMI_PB_Clear_Alarms) ,XIC(Alarm_Word_Current[0].27) ]XIO(System.HMI_PB_Clear_Alarms)XIO(System.Timer_EStop_Reset.TT)[XIC(Alarm_Timer[0,27].DN) OTE(Alarm_Word_Current[0].27) ,TON(Alarm_Timer[0,27],?,?) ];
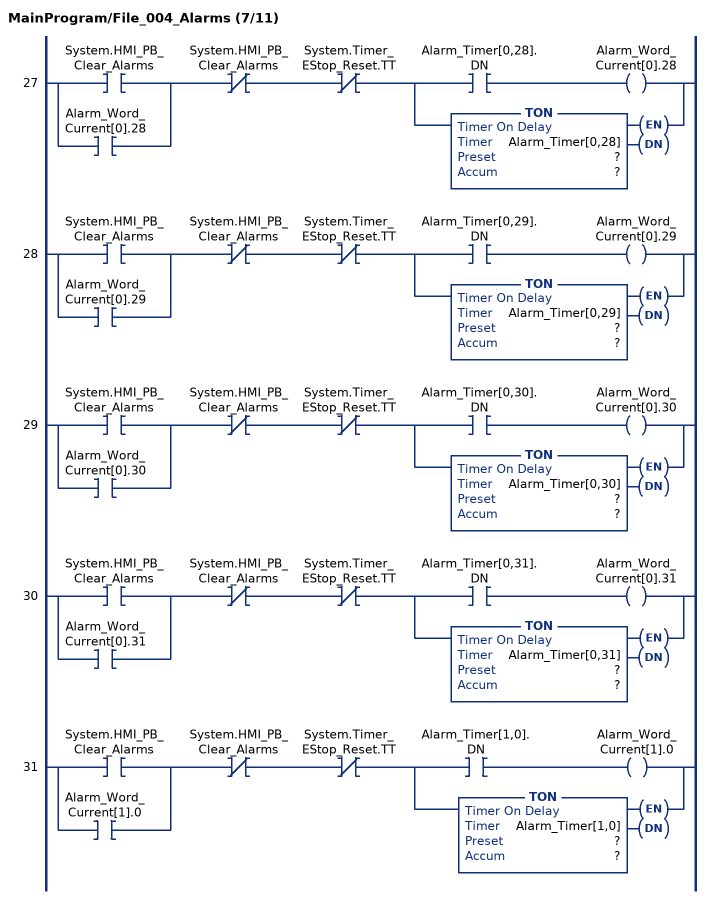
   27: [XIC(System.HMI_PB_Clear_Alarms) ,XIC(Alarm_Word_Current[0].28) ]XIO(System.HMI_PB_Clear_Alarms)XIO(System.Timer_EStop_Reset.TT)[XIC(Alarm_Timer[0,28].DN) OTE(Alarm_Word_Current[0].28) ,TON(Alarm_Timer[0,28],?,?) ];
   28: [XIC(System.HMI_PB_Clear_Alarms) ,XIC(Alarm_Word_Current[0].29) ]XIO(System.HMI_PB_Clear_Alarms)XIO(System.Timer_EStop_Reset.TT)[XIC(Alarm_Timer[0,29].DN) OTE(Alarm_Word_Current[0].29) ,TON(Alarm_Timer[0,29],?,?) ];
   29: [XIC(System.HMI_PB_Clear_Alarms) ,XIC(Alarm_Word_Current[0].30) ]XIO(System.HMI_PB_Clear_Alarms)XIO(System.Timer_EStop_Reset.TT)[XIC(Alarm_Timer[0,30].DN) OTE(Alarm_Word_Current[0].30) ,TON(Alarm_Timer[0,30],?,?) ];
   30: [XIC(System.HMI_PB_Clear_Alarms) ,XIC(Alarm_Word_Current[0].31) ]XIO(System.HMI_PB_Clear_Alarms)XIO(System.Timer_EStop_Reset.TT)[XIC(Alarm_Timer[0,31].DN) OTE(Alarm_Word_Current[0].31) ,TON(Alarm_Timer[0,31],?,?) ];
   31: [XIC(System.HMI_PB_Clear_Alarms) ,XIC(Alarm_Word_Current[1].0) ]XIO(System.HMI_PB_Clear_Alarms)XIO(System.Timer_EStop_Reset.TT)[XIC(Alarm_Timer[1,0].DN) OTE(Alarm_Word_Current[1].0) ,TON(Alarm_Timer[1,0],?,?) ];
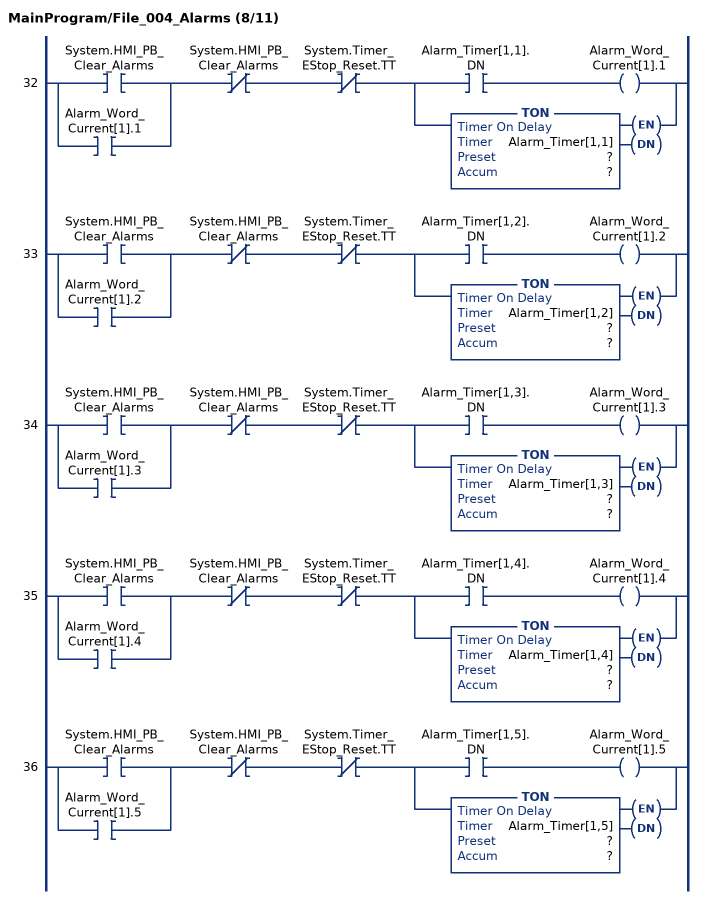
   32: [XIC(System.HMI_PB_Clear_Alarms) ,XIC(Alarm_Word_Current[1].1) ]XIO(System.HMI_PB_Clear_Alarms)XIO(System.Timer_EStop_Reset.TT)[XIC(Alarm_Timer[1,1].DN) OTE(Alarm_Word_Current[1].1) ,TON(Alarm_Timer[1,1],?,?) ];
   33: [XIC(System.HMI_PB_Clear_Alarms) ,XIC(Alarm_Word_Current[1].2) ]XIO(System.HMI_PB_Clear_Alarms)XIO(System.Timer_EStop_Reset.TT)[XIC(Alarm_Timer[1,2].DN) OTE(Alarm_Word_Current[1].2) ,TON(Alarm_Timer[1,2],?,?) ];
   34: [XIC(System.HMI_PB_Clear_Alarms) ,XIC(Alarm_Word_Current[1].3) ]XIO(System.HMI_PB_Clear_Alarms)XIO(System.Timer_EStop_Reset.TT)[XIC(Alarm_Timer[1,3].DN) OTE(Alarm_Word_Current[1].3) ,TON(Alarm_Timer[1,3],?,?) ];
   35: [XIC(System.HMI_PB_Clear_Alarms) ,XIC(Alarm_Word_Current[1].4) ]XIO(System.HMI_PB_Clear_Alarms)XIO(System.Timer_EStop_Reset.TT)[XIC(Alarm_Timer[1,4].DN) OTE(Alarm_Word_Current[1].4) ,TON(Alarm_Timer[1,4],?,?) ];
   36: [XIC(System.HMI_PB_Clear_Alarms) ,XIC(Alarm_Word_Current[1].5) ]XIO(System.HMI_PB_Clear_Alarms)XIO(System.Timer_EStop_Reset.TT)[XIC(Alarm_Timer[1,5].DN) OTE(Alarm_Word_Current[1].5) ,TON(Alarm_Timer[1,5],?,?) ];
